# B&R Automation Studio project Ampel (part 2)

```cpp
	if (request.destination == 0)
		return false;
	else if (HFSM2_CHECKED(request.destination < STATE_COUNT)) {
Parent parent = stateParents[request.destination];

		if (HFSM2_CHECKED(parent)) {
			HFSM2_ASSERT(parent.forkId > 0);

compoRequested[parent.forkId - 1] = parent.prong;

for (parent = forkParent(parent.forkId);
parent;
parent = forkParent(parent.forkId))
			{
				HFSM2_ASSERT(parent.forkId > 0);
				compoRemains.set(parent.forkId - 1);

if (compoActive	  [parent.forkId - 1] != parent.prong)
compoRequested[parent.forkId - 1]  = parent.prong;
				else {
parent = forkParent(parent.forkId);
					break;
				}
			}

for (; parent; parent = forkParent(parent.forkId)) {
				HFSM2_ASSERT(parent.forkId > 0);
				compoRemains.set(parent.forkId - 1);
			}
		}
	}

	return true;
}

template <typename TG_, typename TSL_, typename TRL_, Long NCC_, typename TRO_ HFSM2_IF_SERIALIZATION(, Long NSB_) HFSM2_IF_PLANS(, Long NTC_), typename TTP_>
HFSM2_CONSTEXPR(14)
void
RegistryT<ArgsT<TG_, TSL_, TRL_, NCC_, 0, 0, TRO_ HFSM2_IF_SERIALIZATION(, NSB_) HFSM2_IF_PLANS(, NTC_), TTP_>>::requestScheduled(const StateID stateId) noexcept {
	if (HFSM2_CHECKED(stateId < STATE_COUNT)) {
const Parent parent = stateParents[stateId];

		HFSM2_ASSERT(parent.forkId > 0);
compoResumable[parent.forkId - 1] = parent.prong;
	}
}

template <typename TG_, typename TSL_, typename TRL_, Long NCC_, typename TRO_ HFSM2_IF_SERIALIZATION(, Long NSB_) HFSM2_IF_PLANS(, Long NTC_), typename TTP_>
HFSM2_CONSTEXPR(14)
void
RegistryT<ArgsT<TG_, TSL_, TRL_, NCC_, 0, 0, TRO_ HFSM2_IF_SERIALIZATION(, NSB_) HFSM2_IF_PLANS(, NTC_), TTP_>>::clearRequests() noexcept {
	compoRequested.clear();
	orthoRequested.clear();
	compoRemains  .clear();
}

template <typename TG_, typename TSL_, typename TRL_, Long NCC_, typename TRO_ HFSM2_IF_SERIALIZATION(, Long NSB_) HFSM2_IF_PLANS(, Long NTC_), typename TTP_>
HFSM2_CONSTEXPR(14)
void
RegistryT<ArgsT<TG_, TSL_, TRL_, NCC_, 0, 0, TRO_ HFSM2_IF_SERIALIZATION(, NSB_) HFSM2_IF_PLANS(, NTC_), TTP_>>::clear() noexcept {
	clearRequests();

	compoActive	  .clear();
	compoResumable.clear();
}

template <typename TG_, typename TSL_, typename TRL_, Long NCC_, typename TRO_ HFSM2_IF_SERIALIZATION(, Long NSB_) HFSM2_IF_PLANS(, Long NTC_), typename TTP_>
HFSM2_CONSTEXPR(11)
bool
RegistryT<ArgsT<TG_, TSL_, TRL_, NCC_, 0, 0, TRO_ HFSM2_IF_SERIALIZATION(, NSB_) HFSM2_IF_PLANS(, NTC_), TTP_>>::empty() const noexcept {
	return compoRequested.empty()
		&& orthoRequested.empty()
		&& compoRemains	 .empty()
		&& compoActive	 .empty()
		&& compoResumable.empty();
}

}
}

namespace hfsm2 {
	namespace detail {

		struct TaskStatus final {
		enum Result {
			NONE,
			SUCCESS,
			FAILURE
		};

		Result result = Result::NONE;
		bool outerTransition = false;

		HFSM2_CONSTEXPR(11)	TaskStatus(const Result result_ = Result::NONE,
		const bool outerTransition_ = false)	noexcept;

		HFSM2_CONSTEXPR(11)	explicit operator bool()				  const noexcept;

		HFSM2_CONSTEXPR(14)	void clear()									noexcept;
	};

	HFSM2_CONSTEXPR(14) TaskStatus  operator |  (TaskStatus& l, const TaskStatus r)	noexcept;
	HFSM2_CONSTEXPR(14) TaskStatus& operator |= (TaskStatus& l, const TaskStatus r)	noexcept;

#if HFSM2_PLANS_AVAILABLE()

	struct TaskLink final {
	Long prev		= INVALID_LONG;
	Long next		= INVALID_LONG;
};

struct Bounds final {
Long first		= INVALID_LONG;
Long last		= INVALID_LONG;
};

template <
	typename
  , typename
  , typename
  , Long
  , Long
  , Long
  , typename
  HFSM2_IF_SERIALIZATION(, Long)
, Long
  , typename
>
struct ArgsT;

template <typename>
struct PlanDataT;

template <
	typename TConfig
  , typename TStateList
  , typename TRegionList
  , Long NCompoCount
  , Long NOrthoCount
  , Long NOrthoUnits
  , typename TReactOrder
  HFSM2_IF_SERIALIZATION(, Long NSerialBits)
  , Long NTaskCapacity
  , typename TPayload
>
struct PlanDataT<
	ArgsT<
	TConfig
	, TStateList
	, TRegionList
	, NCompoCount
	, NOrthoCount
	, NOrthoUnits
	, TReactOrder
	HFSM2_IF_SERIALIZATION(, NSerialBits)
	, NTaskCapacity
	, TPayload
	>
	> final
	{
	using StateList			= TStateList;
	using RegionList		= TRegionList;
	using Payload			= TPayload;

	static constexpr Long STATE_COUNT	= StateList ::SIZE;
	static constexpr Long REGION_COUNT	= RegionList::SIZE;
	static constexpr Long TASK_CAPACITY	= NTaskCapacity;

	using Task				= TaskT		  <Payload>;
	using Tasks				= TaskListT   <Payload,  TASK_CAPACITY>;
	using TaskLinks			= StaticArrayT<TaskLink, TASK_CAPACITY>;
	using Payloads			= StaticArrayT<Payload,  TASK_CAPACITY>;

	using TasksBounds		= StaticArrayT<Bounds,	   REGION_COUNT>;
	using TasksBits			= BitArrayT   <				STATE_COUNT>;
	using RegionBits		= BitArrayT   <			   REGION_COUNT>;
	using RegionStatuses	= StaticArrayT<TaskStatus, REGION_COUNT>;

	Tasks tasks;
	TaskLinks taskLinks;
	Payloads taskPayloads;
	TasksBits payloadExists;

	TasksBounds taskBounds;
	TasksBits tasksSuccesses;
	TasksBits tasksFailures;
	RegionBits planExists;
	RegionStatuses headStatuses;
	RegionStatuses subStatuses;

	HFSM2_CONSTEXPR(14)	void clearTaskStatus  (const StateID stateId)		noexcept;
	HFSM2_CONSTEXPR(14)	void verifyEmptyStatus(const StateID stateId) const noexcept;

	HFSM2_CONSTEXPR(14)	void clearStatuses()								noexcept;
	HFSM2_CONSTEXPR(14)	void clear()										noexcept;

#if HFSM2_ASSERT_AVAILABLE()
	HFSM2_CONSTEXPR(14)	void verifyPlans()							  const noexcept;
	HFSM2_CONSTEXPR(14)	Long verifyPlan(const RegionID stateId)		  const noexcept;
#endif
};

template <
	typename TConfig
  , typename TStateList
  , typename TRegionList
  , Long NCompoCount
  , Long NOrthoCount
  , Long NOrthoUnits
  , typename TReactOrder
  HFSM2_IF_SERIALIZATION(, Long NSerialBits)
  , Long NTaskCapacity
>
struct PlanDataT<
		   ArgsT<
			   TConfig
			 , TStateList
			 , TRegionList
			 , NCompoCount
			 , NOrthoCount
			 , NOrthoUnits
			 , TReactOrder
			 HFSM2_IF_SERIALIZATION(, NSerialBits)
			 , NTaskCapacity
			 , void
		   >
	   > final
{
	using StateList			= TStateList;
using RegionList		= TRegionList;

static constexpr Long  STATE_COUNT	= StateList ::SIZE;
static constexpr Long REGION_COUNT	= RegionList::SIZE;
static constexpr Long TASK_CAPACITY	= NTaskCapacity;

	using Task				= TaskT		  <void>;
using Tasks				= TaskListT	  <void,	 TASK_CAPACITY>;
using TaskLinks			= StaticArrayT<TaskLink, TASK_CAPACITY>;

using TasksBounds		= StaticArrayT<Bounds,	   REGION_COUNT>;
using TasksBits			= BitArrayT	  <				STATE_COUNT>;
using RegionBits		= BitArrayT	  <			   REGION_COUNT>;
using RegionStatuses	= StaticArrayT<TaskStatus, REGION_COUNT>;

Tasks tasks;
TaskLinks taskLinks;

TasksBounds taskBounds;
TasksBits tasksSuccesses;
TasksBits tasksFailures;
RegionBits planExists;
RegionStatuses headStatuses;
RegionStatuses subStatuses;

	HFSM2_CONSTEXPR(14)	void clearTaskStatus  (const StateID stateId)		noexcept;
	HFSM2_CONSTEXPR(14)	void verifyEmptyStatus(const StateID stateId) const noexcept;

	HFSM2_CONSTEXPR(14)	void clearStatuses()								noexcept;
	HFSM2_CONSTEXPR(14)	void clear()										noexcept;

#if HFSM2_ASSERT_AVAILABLE()
	HFSM2_CONSTEXPR(14)	void verifyPlans()							  const noexcept;
	HFSM2_CONSTEXPR(14)	Long verifyPlan(const RegionID stateId)		  const noexcept;
#endif
};

template <
	typename TConfig
  , typename TStateList
  , typename TRegionList
  , Long NOrthoCount
  , Long NOrthoUnits
  , typename TReactOrder
  , Long NTaskCapacity
  , typename TPayload
>
struct PlanDataT<
	ArgsT<
	TConfig
	, TStateList
	, TRegionList
	, 0
	, NOrthoCount
	, NOrthoUnits
	, TReactOrder
	HFSM2_IF_SERIALIZATION(, 0)
	, NTaskCapacity
	, TPayload
	>
	> final
	{
HFSM2_CONSTEXPR(14)	void clearTaskStatus  (const StateID)				noexcept	{}
	HFSM2_CONSTEXPR(14)	void verifyEmptyStatus(const StateID)		  const noexcept	{}

	HFSM2_CONSTEXPR(14)	void clearStatuses()								noexcept	{}
	HFSM2_CONSTEXPR(14)	void clear()										noexcept	{}

#if HFSM2_ASSERT_AVAILABLE()
	HFSM2_CONSTEXPR(14)	void verifyPlans()							  const noexcept	{}
#endif
};

template <
	typename TConfig
  , typename TStateList
  , typename TRegionList
  , Long NOrthoCount
  , Long NOrthoUnits
  , typename TReactOrder
  , Long NTaskCapacity
>
struct PlanDataT<
		   ArgsT<
			   TConfig
			 , TStateList
			 , TRegionList
			 , 0
			 , NOrthoCount
			 , NOrthoUnits
			 , TReactOrder
			 HFSM2_IF_SERIALIZATION(, 0)
			 , NTaskCapacity
			 , void
		   >
	   > final
{
	HFSM2_CONSTEXPR(14)	void clearTaskStatus  (const StateID)				noexcept	{}
	HFSM2_CONSTEXPR(14)	void verifyEmptyStatus(const StateID)		  const noexcept	{}

	HFSM2_CONSTEXPR(14)	void clearStatuses()								noexcept	{}
	HFSM2_CONSTEXPR(14)	void clear()										noexcept	{}

#if HFSM2_ASSERT_AVAILABLE()
	HFSM2_CONSTEXPR(14)	void verifyPlans()							  const noexcept	{}
#endif
};

#endif

}
}

namespace hfsm2 {
	namespace detail {

		HFSM2_CONSTEXPR(11)
		TaskStatus::TaskStatus(const Result result_,
		const bool outerTransition_) noexcept
	: result{result_}
, outerTransition{outerTransition_}
{}

HFSM2_CONSTEXPR(11)
TaskStatus::operator bool() const noexcept	{
return result != Result::NONE || outerTransition;
}

HFSM2_CONSTEXPR(14)
void
TaskStatus::clear() noexcept {
result = Result::NONE;
outerTransition = false;
}

HFSM2_CONSTEXPR(14)
TaskStatus
	operator | (TaskStatus& lhs,
	const TaskStatus rhs) noexcept
{
	const TaskStatus::Result result = lhs.result > rhs.result ?
		lhs.result : rhs.result;

	return TaskStatus{result, lhs.outerTransition || rhs.outerTransition};
}

HFSM2_CONSTEXPR(14)
TaskStatus&
	operator |= (TaskStatus& lhs,
	const TaskStatus rhs) noexcept
{
	const TaskStatus::Result result = lhs.result > rhs.result ?
		lhs.result : rhs.result;

	lhs = TaskStatus{result, lhs.outerTransition || rhs.outerTransition};

	return lhs;
}

#if HFSM2_PLANS_AVAILABLE()

template <typename TG_, typename TSL_, typename TRL_, Long NCC_, Long NOC_, Long NOU_, typename TRO_ HFSM2_IF_SERIALIZATION(, Long NSB_), Long NTC_, typename TTP_>
HFSM2_CONSTEXPR(14)
void
	PlanDataT<ArgsT<TG_, TSL_, TRL_, NCC_, NOC_, NOU_, TRO_ HFSM2_IF_SERIALIZATION(, NSB_), NTC_, TTP_>>::clearTaskStatus(const StateID stateId) noexcept {
	if (stateId != INVALID_STATE_ID) {
		tasksSuccesses.clear(stateId);
		tasksFailures .clear(stateId);
	}
}

template <typename TG_, typename TSL_, typename TRL_, Long NCC_, Long NOC_, Long NOU_, typename TRO_ HFSM2_IF_SERIALIZATION(, Long NSB_), Long NTC_, typename TTP_>
HFSM2_CONSTEXPR(14)
void
	PlanDataT<ArgsT<TG_, TSL_, TRL_, NCC_, NOC_, NOU_, TRO_ HFSM2_IF_SERIALIZATION(, NSB_), NTC_, TTP_>>::verifyEmptyStatus(const StateID HFSM2_IF_ASSERT(stateId)) const noexcept {
#if HFSM2_ASSERT_AVAILABLE()

	if (stateId != INVALID_STATE_ID) {
		HFSM2_ASSERT(!tasksSuccesses.get(stateId));
		HFSM2_ASSERT(!tasksFailures .get(stateId));
	}

#endif
}

template <typename TG_, typename TSL_, typename TRL_, Long NCC_, Long NOC_, Long NOU_, typename TRO_ HFSM2_IF_SERIALIZATION(, Long NSB_), Long NTC_, typename TTP_>
HFSM2_CONSTEXPR(14)
void
	PlanDataT<ArgsT<TG_, TSL_, TRL_, NCC_, NOC_, NOU_, TRO_ HFSM2_IF_SERIALIZATION(, NSB_), NTC_, TTP_>>::clearStatuses() noexcept {
	tasksSuccesses.clear();
	tasksFailures .clear();

	headStatuses.clear();
	 subStatuses.clear();
}

template <typename TG_, typename TSL_, typename TRL_, Long NCC_, Long NOC_, Long NOU_, typename TRO_ HFSM2_IF_SERIALIZATION(, Long NSB_), Long NTC_, typename TTP_>
HFSM2_CONSTEXPR(14)
void
	PlanDataT<ArgsT<TG_, TSL_, TRL_, NCC_, NOC_, NOU_, TRO_ HFSM2_IF_SERIALIZATION(, NSB_), NTC_, TTP_>>::clear() noexcept {
	tasks		 .clear();
	taskLinks	 .clear();
	taskPayloads .clear();
	payloadExists.clear();

	taskBounds	 .clear();
	planExists	 .clear();

	clearStatuses();
}

#if HFSM2_ASSERT_AVAILABLE()

template <typename TG_, typename TSL_, typename TRL_, Long NCC_, Long NOC_, Long NOU_, typename TRO_ HFSM2_IF_SERIALIZATION(, Long NSB_), Long NTC_, typename TTP_>
HFSM2_CONSTEXPR(14)
void
	PlanDataT<ArgsT<TG_, TSL_, TRL_, NCC_, NOC_, NOU_, TRO_ HFSM2_IF_SERIALIZATION(, NSB_), NTC_, TTP_>>::verifyPlans() const noexcept {
Long planCount = 0;

for (RegionID regionId = 0; regionId < REGION_COUNT; ++regionId)
		planCount += verifyPlan(regionId);

	HFSM2_ASSERT(tasks.count() == planCount);
}

template <typename TG_, typename TSL_, typename TRL_, Long NCC_, Long NOC_, Long NOU_, typename TRO_ HFSM2_IF_SERIALIZATION(, Long NSB_), Long NTC_, typename TTP_>
HFSM2_CONSTEXPR(14)
Long
	PlanDataT<ArgsT<TG_, TSL_, TRL_, NCC_, NOC_, NOU_, TRO_ HFSM2_IF_SERIALIZATION(, NSB_), NTC_, TTP_>>::verifyPlan(const RegionID regionId) const noexcept {
Long length = 0;
const Bounds& bounds = taskBounds[regionId];

	if (bounds.first != INVALID_LONG) {
		HFSM2_ASSERT(bounds.last != INVALID_LONG);

for (Long slow = bounds.first, fast = slow; ; ) {
++length;
const TaskLink& task = taskLinks[slow];

			if (slow != bounds.last) {
				HFSM2_ASSERT(task.next != INVALID_LONG);
slow = task.next;

				// loop check
				if (fast != INVALID_LONG) {
fast = taskLinks[fast].next;

					if (fast != INVALID_LONG)
fast = taskLinks[fast].next;

					HFSM2_ASSERT(fast == INVALID_LONG || slow != fast);
				}
			} else {
				HFSM2_ASSERT(task.next == INVALID_LONG);

				break;
			}
		};
	} else
		HFSM2_ASSERT(bounds.last == INVALID_LONG);

return length;
}

#endif

template <typename TG_, typename TSL_, typename TRL_, Long NCC_, Long NOC_, Long NOU_, typename TRO_ HFSM2_IF_SERIALIZATION(, Long NSB_), Long NTC_>
HFSM2_CONSTEXPR(14)
void
PlanDataT<ArgsT<TG_, TSL_, TRL_, NCC_, NOC_, NOU_, TRO_ HFSM2_IF_SERIALIZATION(, NSB_), NTC_, void>>::clearTaskStatus(const StateID stateId) noexcept {
	if (stateId != INVALID_STATE_ID) {
		tasksSuccesses.clear(stateId);
		tasksFailures .clear(stateId);
	}
}

template <typename TG_, typename TSL_, typename TRL_, Long NCC_, Long NOC_, Long NOU_, typename TRO_ HFSM2_IF_SERIALIZATION(, Long NSB_), Long NTC_>
HFSM2_CONSTEXPR(14)
void
PlanDataT<ArgsT<TG_, TSL_, TRL_, NCC_, NOC_, NOU_, TRO_ HFSM2_IF_SERIALIZATION(, NSB_), NTC_, void>>::verifyEmptyStatus(const StateID HFSM2_IF_ASSERT(stateId)) const noexcept {
#if HFSM2_ASSERT_AVAILABLE()

	if (stateId != INVALID_STATE_ID) {
		HFSM2_ASSERT(!tasksSuccesses.get(stateId));
		HFSM2_ASSERT(!tasksFailures .get(stateId));
	}

#endif
}

template <typename TG_, typename TSL_, typename TRL_, Long NCC_, Long NOC_, Long NOU_, typename TRO_ HFSM2_IF_SERIALIZATION(, Long NSB_), Long NTC_>
HFSM2_CONSTEXPR(14)
void
PlanDataT<ArgsT<TG_, TSL_, TRL_, NCC_, NOC_, NOU_, TRO_ HFSM2_IF_SERIALIZATION(, NSB_), NTC_, void>>::clearStatuses() noexcept {
	tasksSuccesses.clear();
	tasksFailures .clear();

	headStatuses.clear();
	 subStatuses.clear();
}

template <typename TG_, typename TSL_, typename TRL_, Long NCC_, Long NOC_, Long NOU_, typename TRO_ HFSM2_IF_SERIALIZATION(, Long NSB_), Long NTC_>
HFSM2_CONSTEXPR(14)
void
PlanDataT<ArgsT<TG_, TSL_, TRL_, NCC_, NOC_, NOU_, TRO_ HFSM2_IF_SERIALIZATION(, NSB_), NTC_, void>>::clear() noexcept {
	tasks	  .clear();
	taskLinks .clear();

	taskBounds.clear();
	planExists.clear();

	clearStatuses();
}

#if HFSM2_ASSERT_AVAILABLE()

template <typename TG_, typename TSL_, typename TRL_, Long NCC_, Long NOC_, Long NOU_, typename TRO_ HFSM2_IF_SERIALIZATION(, Long NSB_), Long NTC_>
HFSM2_CONSTEXPR(14)
void
PlanDataT<ArgsT<TG_, TSL_, TRL_, NCC_, NOC_, NOU_, TRO_ HFSM2_IF_SERIALIZATION(, NSB_), NTC_, void>>::verifyPlans() const noexcept {
Long planCount = 0;

for (RegionID regionId = 0; regionId < REGION_COUNT; ++regionId)
		planCount += verifyPlan(regionId);

	HFSM2_ASSERT(tasks.count() == planCount);
}

template <typename TG_, typename TSL_, typename TRL_, Long NCC_, Long NOC_, Long NOU_, typename TRO_ HFSM2_IF_SERIALIZATION(, Long NSB_), Long NTC_>
HFSM2_CONSTEXPR(14)
Long
PlanDataT<ArgsT<TG_, TSL_, TRL_, NCC_, NOC_, NOU_, TRO_ HFSM2_IF_SERIALIZATION(, NSB_), NTC_, void>>::verifyPlan(const RegionID regionId) const noexcept {
Long length = 0;
const Bounds& bounds = taskBounds[regionId];

	if (bounds.first != INVALID_LONG) {
		HFSM2_ASSERT(bounds.last != INVALID_LONG);

for (auto slow = bounds.first, fast = slow; ; ) {
++length;
const TaskLink& task = taskLinks[slow];

			if (slow != bounds.last) {
				HFSM2_ASSERT(task.next != INVALID_LONG);
slow = task.next;

				// loop check
				if (fast != INVALID_LONG) {
fast = taskLinks[fast].next;

					if (fast != INVALID_LONG)
fast = taskLinks[fast].next;

					HFSM2_ASSERT(fast == INVALID_LONG || slow != fast);
				}
			} else {
				HFSM2_ASSERT(task.next == INVALID_LONG);

				break;
			}
		};
	} else
		HFSM2_ASSERT(bounds.last == INVALID_LONG);

return length;
}

#endif
#endif

}
}

#if HFSM2_PLANS_AVAILABLE()

namespace hfsm2 {
	namespace detail {

		template <typename TArgs>
		class CPlanT {
			template <typename>
			friend class ControlT;

			template <typename>
			friend class PlanControlT;

			template <typename>
			friend class FullControlT;

			template <typename>
			friend class GuardControlT;

			template <typename, typename>
			friend class R_;

			using Args			= TArgs;
			using Context		= typename Args::Context;
			using StateList		= typename Args::StateList;
			using RegionList	= typename Args::RegionList;

			static constexpr Long TASK_CAPACITY = Args::TASK_CAPACITY;

			public:
			using PlanData		= PlanDataT<Args>;
			using Task			= typename PlanData::Task;
			using TaskLinks		= typename PlanData::TaskLinks;

			struct Iterator final {
			HFSM2_CONSTEXPR(14)	Iterator(const CPlanT& plan)				noexcept;

			HFSM2_CONSTEXPR(14)	explicit operator bool()			  const noexcept;

			HFSM2_CONSTEXPR(14)	void operator ++()							noexcept;

			HFSM2_CONSTEXPR(11)	bool operator != (const Iterator)	  const noexcept	{ return operator bool();					}

			HFSM2_CONSTEXPR(11)	const Task& operator  *()			  const noexcept	{ return  _plan._planData.tasks[_curr];		}
			HFSM2_CONSTEXPR(11)	const Task* operator ->()			  const noexcept	{ return &_plan._planData.tasks[_curr];		}

			HFSM2_CONSTEXPR(14)	Long next()							  const noexcept;

			const CPlanT& _plan;
			Long _curr;
			Long _next;
		};

		private:
		HFSM2_CONSTEXPR(11)	CPlanT(const PlanData& planData,
		const RegionID regionId_)				noexcept
	: _planData{planData}
, _bounds{planData.taskBounds[regionId_]}
	{}

	template <typename TState>
	static
	HFSM2_CONSTEXPR(11)  StateID  stateId()								noexcept	{ return					   index<StateList , TState>();		}

	template <typename TState>
	static
	HFSM2_CONSTEXPR(11)	RegionID regionId()								noexcept	{ return static_cast<RegionID>(index<RegionList, TState>());	}

public:
	HFSM2_CONSTEXPR(14)	explicit operator bool()				  const noexcept;

	/// @brief Begin iteration over plan tasks
	/// @return CIterator to the first task
	HFSM2_CONSTEXPR(14)	Iterator begin()								noexcept	{ return Iterator{*this};					}

	/// @brief Iteration terminator
	/// @return Dummy Iterator
	HFSM2_CONSTEXPR(14)	Iterator end  ()								noexcept	{ return Iterator{*this};					}

	/// @brief First task
	/// @return First task
	HFSM2_CONSTEXPR(14) const Task& first()						  const noexcept;

	/// @brief Last task
	/// @return Last task
	HFSM2_CONSTEXPR(14) const Task&  last()						  const noexcept;

private:
const PlanData& _planData;
const Bounds& _bounds;
};

}
}

#endif

#if HFSM2_PLANS_AVAILABLE()

namespace hfsm2 {
	namespace detail {

		template <typename TArgs>
		HFSM2_CONSTEXPR(14)
		CPlanT<TArgs>::Iterator::Iterator(const CPlanT& plan) noexcept
	: _plan{plan}
, _curr{plan._bounds.first}
{
	_next = next();
}

template <typename TArgs>
HFSM2_CONSTEXPR(14)
CPlanT<TArgs>::Iterator::operator bool() const noexcept {
	HFSM2_ASSERT(_curr < CPlanT::TASK_CAPACITY ||
				 _curr == INVALID_LONG);

return _curr < CPlanT::TASK_CAPACITY;
}

template <typename TArgs>
HFSM2_CONSTEXPR(14)
void
CPlanT<TArgs>::Iterator::operator ++() noexcept {
	_curr = _next;
	_next = next();
}

template <typename TArgs>
HFSM2_CONSTEXPR(14)
Long
CPlanT<TArgs>::Iterator::next() const noexcept {
	if (_curr < CPlanT::TASK_CAPACITY) {
		const TaskLink& link = _plan._planData.taskLinks[_curr];

		return link.next;
	} else {
		HFSM2_ASSERT(_curr == INVALID_LONG);

		return INVALID_LONG;
	}
}

template <typename TArgs>
HFSM2_CONSTEXPR(14)
CPlanT<TArgs>::operator bool() const noexcept {
	HFSM2_ASSERT(_bounds.first < TASK_CAPACITY &&
				 _bounds.last  < TASK_CAPACITY ||
				 _bounds.last == INVALID_LONG);

return _bounds.first < TASK_CAPACITY;
}

template <typename TArgs>
HFSM2_CONSTEXPR(14)
const typename CPlanT<TArgs>::Task&
CPlanT<TArgs>::first() const noexcept {
	HFSM2_ASSERT(_bounds.first < TASK_CAPACITY);

	return _planData.tasks[_bounds.first];
}

template <typename TArgs>
HFSM2_CONSTEXPR(14)
const typename CPlanT<TArgs>::Task&
CPlanT<TArgs>::last() const noexcept {
	HFSM2_ASSERT(_bounds.last < TASK_CAPACITY);

	return _planData.tasks[_bounds.last];
}

}
}

#endif

#if HFSM2_PLANS_AVAILABLE()

namespace hfsm2 {
	namespace detail {

		template <typename TArgs>
		class PlanT {
			template <typename, typename, Strategy, typename, typename...>
			friend struct C_;

			template <typename, typename, typename, typename...>
			friend struct O_;

			using Args			= TArgs;
			using Context		= typename Args::Context;
			using StateList		= typename Args::StateList;
			using RegionList	= typename Args::RegionList;

			using Registry		= RegistryT<Args>;

			static constexpr Long  TASK_CAPACITY	= Args::TASK_CAPACITY;

			public:
			using PlanData		= PlanDataT<Args>;
			using Task			= typename PlanData::Task;
			using Tasks			= typename PlanData::Tasks;
			using TaskLinks		= typename PlanData::TaskLinks;
			using TaskIndex		= typename TaskLinks::Index;
			using TasksBits		= typename PlanData::TasksBits;

			struct CIterator final {
			HFSM2_CONSTEXPR(14)	CIterator(const PlanT& plan)				noexcept;

			HFSM2_CONSTEXPR(14)	explicit operator bool()			  const noexcept;

			HFSM2_CONSTEXPR(14)	void operator ++()							noexcept;

			HFSM2_CONSTEXPR(14)	bool operator != (const CIterator)	  const noexcept	{ return operator bool();					}

			HFSM2_CONSTEXPR(14)	const Task& operator  *()			  const noexcept	{ return  _plan._planData.tasks[_curr];		}
			HFSM2_CONSTEXPR(11)	const Task* operator ->()			  const noexcept	{ return &_plan._planData.tasks[_curr];		}

			HFSM2_CONSTEXPR(14)	Long next()							  const noexcept;

			const PlanT& _plan;
			Long _curr;
			Long _next;
		};

		struct Iterator final {
		HFSM2_CONSTEXPR(14)	Iterator(PlanT& plan)						noexcept;

		HFSM2_CONSTEXPR(14)	explicit operator bool()			  const noexcept;

		HFSM2_CONSTEXPR(14)	void operator ++()							noexcept;

		HFSM2_CONSTEXPR(14)	bool operator != (const Iterator)	  const noexcept	{ return operator bool();					}

		HFSM2_CONSTEXPR(14)	Task& operator  *()							noexcept	{ return  _plan._planData.tasks[_curr];		}
		HFSM2_CONSTEXPR(14)	Task* operator ->()							noexcept	{ return &_plan._planData.tasks[_curr];		}

	HFSM2_CONSTEXPR(14)	void remove()								noexcept	{ _plan.remove(_curr);						}

	HFSM2_CONSTEXPR(14)	Long next()							  const noexcept;

	PlanT& _plan;
	Long _curr;
	Long _next;
};

protected:
	HFSM2_CONSTEXPR(11)	PlanT(Registry& registry,
							  PlanData& planData,
							  const RegionID regionId_)					noexcept;

	template <typename TState>
	static
	HFSM2_CONSTEXPR(11)  StateID  stateId()								noexcept	{ return					   index<StateList , TState>();		}

	template <typename TState>
	static
	HFSM2_CONSTEXPR(11) RegionID regionId()								noexcept	{ return static_cast<RegionID>(index<RegionList, TState>());	}

	HFSM2_CONSTEXPR(14)	bool  append(const StateID origin,
									 const StateID destination,
									 const TransitionType type)			noexcept;

	HFSM2_CONSTEXPR(14)	bool linkTask(const Long index)					noexcept;

	HFSM2_CONSTEXPR(14)	void clearTasks()								noexcept;
	HFSM2_CONSTEXPR(14)	void clearStatuses()							noexcept;

public:
	HFSM2_CONSTEXPR(14)	explicit operator bool()				  const noexcept;

	/// @brief Clear all tasks from the plan
	HFSM2_CONSTEXPR(14)	void clear()									noexcept;

	/// @brief Append a task to transition from `origin` to `destination` if `origin` completes with `success()`
	///   (if transitioning into a region, acts depending on the region type)
	/// @param `origin` Origin state identifier
	/// @param `destination` Destination state identifier
	/// @return Seccess if FSM total number of tasks is below task capacity
	/// @note use `Config::TaskCapacityN<>` to increase task capacity if necessary
	HFSM2_CONSTEXPR(14)	bool change   (const StateID origin,
									   const StateID destination)		noexcept	{ return append	  (origin, destination, TransitionType::CHANGE	 );	}

	/// @brief Append a task to transition from `origin` to `destination` if `origin` completes with `success()`
	///   (if transitioning into a region, acts depending on the region type)
	/// @tparam `TOrigin` Origin state type
	/// @param `destination` Destination state identifier
	/// @return Seccess if FSM total number of tasks is below task capacity
	/// @note use `Config::TaskCapacityN<>` to increase task capacity if necessary
	template <typename TOrigin>
	HFSM2_CONSTEXPR(14)	bool change   (const StateID destination)		noexcept	{ return change	  (stateId<TOrigin>() , destination				 );	}

	/// @brief Append a task to transition from `origin` to `destination` if `origin` completes with `success()`
	///   (if transitioning into a region, acts depending on the region type)
	/// @tparam `TOrigin` Origin state type
	/// @tparam `TDestination` Destination state type
	/// @return Seccess if FSM total number of tasks is below task capacity
	/// @note use `Config::TaskCapacityN<>` to increase task capacity if necessary
	template <typename TOrigin, typename TDestination>
	HFSM2_CONSTEXPR(14)	bool change   ()								noexcept	{ return change	  (stateId<TOrigin>() , stateId<TDestination>()	 );	}

	/// @brief Append a task to transition from `origin` to `destination` if `origin` completes with `success()`
	///   (if transitioning into a region, activates the initial state)
	/// @tparam `TOrigin` Origin state type
	/// @param `destination` Destination state identifier
	/// @return Seccess if FSM total number of tasks is below task capacity
	/// @note use `Config::TaskCapacityN<>` to increase task capacity if necessary
	HFSM2_CONSTEXPR(14)	bool restart  (const StateID origin,
									   const StateID destination)		noexcept	{ return append	  (origin, destination, TransitionType::RESTART	 );	}

	/// @brief Append a task to transition from `origin` to `destination` if `origin` completes with `success()`
	///   (if transitioning into a region, activates the initial state)
	/// @tparam `TOrigin` Origin state type
	/// @param `destination` Destination state identifier
	/// @return Seccess if FSM total number of tasks is below task capacity
	/// @note use `Config::TaskCapacityN<>` to increase task capacity if necessary
	template <typename TOrigin>
	HFSM2_CONSTEXPR(14)	bool restart  (const StateID destination)		noexcept	{ return restart  (stateId<TOrigin>() , destination				 );	}

	/// @brief Append a task to transition from `origin` to `destination` if `origin` completes with `success()`
	///   (if transitioning into a region, activates the initial state)
	/// @tparam `TOrigin` Origin state type
	/// @tparam `TDestination` Destination state type
	/// @return Seccess if FSM total number of tasks is below task capacity
	/// @note use `Config::TaskCapacityN<>` to increase task capacity if necessary
	template <typename TOrigin, typename TDestination>
	HFSM2_CONSTEXPR(14)	bool restart  ()								noexcept	{ return restart  (stateId<TOrigin>() , stateId<TDestination>()	 );	}

	/// @brief Append a task to transition from `origin` to `destination` if `origin` completes with `success()`
	///   (if transitioning into a region, activates the state that was active previously)
	/// @tparam `TOrigin` Origin state type
	/// @param `destination` Destination state identifier
	/// @return Seccess if FSM total number of tasks is below task capacity
	/// @note use `Config::TaskCapacityN<>` to increase task capacity if necessary
	HFSM2_CONSTEXPR(14)	bool resume   (const StateID origin,
									   const StateID destination)		noexcept	{ return append	  (origin, destination, TransitionType::RESUME	 );	}

	/// @brief Append a task to transition from `origin` to `destination` if `origin` completes with `success()`
	///   (if transitioning into a region, activates the state that was active previously)
	/// @tparam `TOrigin` Origin state type
	/// @param `destination` Destination state identifier
	/// @return Seccess if FSM total number of tasks is below task capacity
	/// @note use `Config::TaskCapacityN<>` to increase task capacity if necessary
	template <typename TOrigin>
	HFSM2_CONSTEXPR(14)	bool resume   (const StateID destination)		noexcept	{ return resume	  (stateId<TOrigin>() , destination				 );	}

	/// @brief Append a task to transition from `origin` to `destination` if `origin` completes with `success()`
	///   (if transitioning into a region, activates the state that was active previously)
	/// @tparam `TOrigin` Origin state type
	/// @tparam `TDestination` Destination state type
	/// @return Seccess if FSM total number of tasks is below task capacity
	/// @note use `Config::TaskCapacityN<>` to increase task capacity if necessary
	template <typename TOrigin, typename TDestination>
	HFSM2_CONSTEXPR(14)	bool resume   ()								noexcept	{ return resume	  (stateId<TOrigin>() , stateId<TDestination>()	 );	}

	/// @brief Append a task to transition from `origin` to `destination` if `origin` completes with `success()`
	///   (if transitioning into a region, activates the sub-state by index returned by the region's `select()` method)
	/// @tparam `TOrigin` Origin state type
	/// @param `destination` Destination state identifier
	/// @return Seccess if FSM total number of tasks is below task capacity
	/// @note use `Config::TaskCapacityN<>` to increase task capacity if necessary
	HFSM2_CONSTEXPR(14)	bool select   (const StateID origin,
									   const StateID destination)		noexcept	{ return append	  (origin, destination, TransitionType::SELECT	 );	}

	/// @brief Append a task to transition from `origin` to `destination` if `origin` completes with `success()`
	///   (if transitioning into a region, activates the sub-state by index returned by the region's `select()` method)
	/// @tparam `TOrigin` Origin state type
	/// @param `destination` Destination state identifier
	/// @return Seccess if FSM total number of tasks is below task capacity
	/// @note use `Config::TaskCapacityN<>` to increase task capacity if necessary
	template <typename TOrigin>
	HFSM2_CONSTEXPR(14)	bool select   (const StateID destination)		noexcept	{ return select	  (stateId<TOrigin>() , destination				 );	}

	/// @brief Append a task to transition from `origin` to `destination` if `origin` completes with `success()`
	///   (if transitioning into a region, activates the sub-state by index returned by the region's `select()` method)
	/// @tparam `TOrigin` Origin state type
	/// @tparam `TDestination` Destination state type
	/// @return Seccess if FSM total number of tasks is below task capacity
	/// @note use `Config::TaskCapacityN<>` to increase task capacity if necessary
	template <typename TOrigin, typename TDestination>
	HFSM2_CONSTEXPR(14)	bool select   ()								noexcept	{ return select	  (stateId<TOrigin>() , stateId<TDestination>()	 );	}

#if HFSM2_UTILITY_THEORY_AVAILABLE()

	/// @brief Append a task to transition from `origin` to `destination` if `origin` completes with `success()`
	///   (if transitioning into a region, activates the state with the highest `utility()`
	///   among those with the highest `rank()`)
	/// @tparam `TOrigin` Origin state type
	/// @param `destination` Destination state identifier
	/// @return Seccess if FSM total number of tasks is below task capacity
	/// @note use `Config::TaskCapacityN<>` to increase task capacity if necessary
	/// @see `HFSM2_ENABLE_UTILITY_THEORY`
	HFSM2_CONSTEXPR(14)	bool utilize  (const StateID origin,
									   const StateID destination)		noexcept	{ return append	  (origin, destination, TransitionType::UTILIZE	 );	}

	/// @brief Append a task to transition from `origin` to `destination` if `origin` completes with `success()`
	///   (if transitioning into a region, activates the state with the highest `utility()`
	///   among those with the highest `rank()`)
	/// @tparam `TOrigin` Origin state type
	/// @param `destination` Destination state identifier
	/// @return Seccess if FSM total number of tasks is below task capacity
	/// @note use `Config::TaskCapacityN<>` to increase task capacity if necessary
	/// @see `HFSM2_ENABLE_UTILITY_THEORY`
	template <typename TOrigin>
	HFSM2_CONSTEXPR(14)	bool utilize  (const StateID destination)		noexcept	{ return utilize  (stateId<TOrigin>() , destination				 );	}

	/// @brief Append a task to transition from `origin` to `destination` if `origin` completes with `success()`
	///   (if transitioning into a region, activates the state with the highest `utility()`
	///   among those with the highest `rank()`)
	/// @tparam `TOrigin` Origin state type
	/// @tparam `TDestination` Destination state type
	/// @return Seccess if FSM total number of tasks is below task capacity
	/// @note use `Config::TaskCapacityN<>` to increase task capacity if necessary
	/// @see `HFSM2_ENABLE_UTILITY_THEORY`
	template <typename TOrigin, typename TDestination>
	HFSM2_CONSTEXPR(14)	bool utilize  ()								noexcept	{ return utilize  (stateId<TOrigin>() , stateId<TDestination>()	 );	}

	/// @brief Append a task to transition from `origin` to `destination` if `origin` completes with `success()`
	///   (if transitioning into a region, uses weighted random to activate the state proportional to `utility()`
	///   among those with the highest `rank()`)
	/// @tparam `TOrigin` Origin state type
	/// @param `destination` Destination state identifier
	/// @return Seccess if FSM total number of tasks is below task capacity
	/// @note use `Config::TaskCapacityN<>` to increase task capacity if necessary
	/// @see `HFSM2_ENABLE_UTILITY_THEORY`
	HFSM2_CONSTEXPR(14)	bool randomize(const StateID origin,
									   const StateID destination)		noexcept	{ return append	  (origin, destination, TransitionType::RANDOMIZE);	}

	/// @brief Append a task to transition from `origin` to `destination` if `origin` completes with `success()`
	///   (if transitioning into a region, uses weighted random to activate the state proportional to `utility()`
	///   among those with the highest `rank()`)
	/// @tparam `TOrigin` Origin state type
	/// @param `destination` Destination state identifier
	/// @return Seccess if FSM total number of tasks is below task capacity
	/// @note use `Config::TaskCapacityN<>` to increase task capacity if necessary
	/// @see `HFSM2_ENABLE_UTILITY_THEORY`
	template <typename TOrigin>
	HFSM2_CONSTEXPR(14)	bool randomize(const StateID destination)		noexcept	{ return randomize(stateId<TOrigin>() , destination				 );	}

	/// @brief Append a task to transition from `origin` to `destination` if `origin` completes with `success()`
	///   (if transitioning into a region, uses weighted random to activate the state proportional to `utility()`
	///   among those with the highest `rank()`)
	/// @tparam `TOrigin` Origin state type
	/// @tparam `TDestination` Destination state type
	/// @return Seccess if FSM total number of tasks is below task capacity
	/// @note use `Config::TaskCapacityN<>` to increase task capacity if necessary
	/// @see `HFSM2_ENABLE_UTILITY_THEORY`
	template <typename TOrigin, typename TDestination>
	HFSM2_CONSTEXPR(14)	bool randomize()								noexcept	{ return randomize(stateId<TOrigin>() , stateId<TDestination>()	 );	}

#endif

	/// @brief Append a task to schedule a transition to `destination` if `origin` completes with `success()`
	/// @tparam `TOrigin` Origin state type
	/// @param `destination` Destination state identifier
	/// @return Seccess if FSM total number of tasks is below task capacity
	/// @note use `Config::TaskCapacityN<>` to increase task capacity if necessary
	HFSM2_CONSTEXPR(14)	bool schedule (const StateID origin,
									   const StateID destination)		noexcept	{ return append	  (origin, destination, TransitionType::SCHEDULE );	}

	/// @brief Append a task to schedule a transition to `destination` if `origin` completes with `success()`
	/// @tparam `TOrigin` Origin state type
	/// @param `destination` Destination state identifier
	/// @return Seccess if FSM total number of tasks is below task capacity
	/// @note use `Config::TaskCapacityN<>` to increase task capacity if necessary
	template <typename TOrigin>
	HFSM2_CONSTEXPR(14)	bool schedule (const StateID destination)		noexcept	{ return schedule (stateId<TOrigin>() , destination				 );	}

	/// @brief Append a task to schedule a transition to `destination` if `origin` completes with `success()`
	/// @tparam `TOrigin` Origin state type
	/// @tparam `TDestination` Destination state type
	/// @return Seccess if FSM total number of tasks is below task capacity
	/// @note use `Config::TaskCapacityN<>` to increase task capacity if necessary
	template <typename TOrigin, typename TDestination>
	HFSM2_CONSTEXPR(14)	bool schedule ()								noexcept	{ return schedule (stateId<TOrigin>() , stateId<TDestination>()	 );	}

	/// @brief Begin iteration over plan tasks
	/// @return Iterator to the first task
	HFSM2_CONSTEXPR(14)	 Iterator begin()								noexcept	{ return  Iterator{*this};	}

	/// @brief Begin iteration over plan tasks
	/// @return CIterator to the first task
	HFSM2_CONSTEXPR(11)	CIterator begin()						  const noexcept	{ return CIterator{*this};	}

private:
	HFSM2_CONSTEXPR(14)	void remove(const Long task)					noexcept;

protected:
Registry& _registry;
PlanData& _planData;
const RegionID _regionId;
Bounds& _bounds;
};

}
}

#endif

#if HFSM2_PLANS_AVAILABLE()

namespace hfsm2 {
	namespace detail {

		template <typename TArgs>
		HFSM2_CONSTEXPR(14)
		PlanT<TArgs>::CIterator::CIterator(const PlanT& plan) noexcept
	: _plan{plan}
, _curr{plan._bounds.first}
	, _next{next()}
{}

template <typename TArgs>
HFSM2_CONSTEXPR(14)
PlanT<TArgs>::CIterator::operator bool() const noexcept {
	HFSM2_ASSERT(_curr  < PlanT::TASK_CAPACITY ||
				 _curr == INVALID_LONG);

return _curr < PlanT::TASK_CAPACITY;
}

template <typename TArgs>
HFSM2_CONSTEXPR(14)
void
PlanT<TArgs>::CIterator::operator ++() noexcept {
	_curr = _next;
	_next = next();
}

template <typename TArgs>
HFSM2_CONSTEXPR(14)
Long
PlanT<TArgs>::CIterator::next() const noexcept {
	if (_curr < PlanT::TASK_CAPACITY) {
		const TaskLink& link = _plan._planData.taskLinks[_curr];

		return link.next;
	} else {
		HFSM2_ASSERT(_curr == INVALID_LONG);

		return INVALID_LONG;
	}
}

template <typename TArgs>
HFSM2_CONSTEXPR(14)
PlanT<TArgs>::Iterator::Iterator(PlanT& plan) noexcept
	: _plan{plan}
	, _curr{plan._bounds.first}
	, _next{next()}
{}

template <typename TArgs>
HFSM2_CONSTEXPR(14)
PlanT<TArgs>::Iterator::operator bool() const noexcept {
	HFSM2_ASSERT(_curr < PlanT::TASK_CAPACITY ||
				 _curr == INVALID_LONG);

return _curr < PlanT::TASK_CAPACITY;
}

template <typename TArgs>
HFSM2_CONSTEXPR(14)
void
PlanT<TArgs>::Iterator::operator ++() noexcept {
	_curr = _next;
	_next = next();
}

template <typename TArgs>
HFSM2_CONSTEXPR(14)
Long
PlanT<TArgs>::Iterator::next() const noexcept {
	if (_curr < PlanT::TASK_CAPACITY) {
		const TaskLink& link = _plan._planData.taskLinks[_curr];

		return link.next;
	} else {
		HFSM2_ASSERT(_curr == INVALID_LONG);

		return INVALID_LONG;
	}
}

template <typename TArgs>
HFSM2_CONSTEXPR(11)
PlanT<TArgs>::PlanT(Registry& registry,
					PlanData& planData,
					const RegionID regionId_) noexcept
	: _registry{registry}
	, _planData{planData}
	, _regionId{regionId_}
, _bounds{planData.taskBounds[regionId_]}
{}

template <typename TArgs>
HFSM2_CONSTEXPR(14)
bool
PlanT<TArgs>:: append(const StateID origin,
					  const StateID destination,
					  const TransitionType type) noexcept
{
	if (_planData.tasks.count() < TASK_CAPACITY) {
		_planData.planExists.set(_regionId);

		return linkTask(_planData.tasks.emplace(origin, destination, type));
	} else
		return false;
}

template <typename TArgs>
HFSM2_CONSTEXPR(14)
bool
PlanT<TArgs>::linkTask(const Long index) noexcept {
	if (index != Tasks::INVALID) {
		if (_bounds.first == INVALID_LONG) {
			HFSM2_ASSERT(_bounds.last == INVALID_LONG);
			HFSM2_ASSERT(_planData.taskLinks[index].prev == INVALID_LONG);
			HFSM2_ASSERT(_planData.taskLinks[index].next == INVALID_LONG);

_bounds.first = index;
_bounds.last  = index;
		} else {
			HFSM2_ASSERT(_bounds.first < TaskLinks::CAPACITY);
			HFSM2_ASSERT(_bounds.last  < TaskLinks::CAPACITY);

TaskLink& lastLink = _planData.taskLinks[_bounds.last];
			HFSM2_ASSERT(lastLink.next == INVALID_LONG);

lastLink.next  = index;

TaskLink& currLink = _planData.taskLinks[index];
			HFSM2_ASSERT(currLink.prev == INVALID_LONG);

currLink.prev  = _bounds.last;

_bounds.last   = index;
		}

		return true;
	} else
		return false;
}

template <typename TArgs>
HFSM2_CONSTEXPR(14)
void
PlanT<TArgs>::clearTasks() noexcept {
	if (_bounds.first < TaskLinks::CAPACITY) {
		HFSM2_ASSERT(_bounds.last < TaskLinks::CAPACITY);

for (Long index = _bounds.first;
index != INVALID_LONG;
			 )
		{
			HFSM2_ASSERT(index < TaskLinks::CAPACITY);

const TaskLink& link = _planData.taskLinks[index];
			HFSM2_ASSERT(index == _bounds.first ?
							 link.prev == INVALID_LONG :
							 link.prev <  TaskLinks::CAPACITY);

const Long next = link.next;

			remove(index);

index = next;
		}

_bounds.first = INVALID_LONG;
_bounds.last  = INVALID_LONG;
	} else {
		HFSM2_ASSERT(_bounds.first == INVALID_LONG);
		HFSM2_ASSERT(_bounds.last  == INVALID_LONG);
	}
}

template <typename TArgs>
HFSM2_CONSTEXPR(14)
void
PlanT<TArgs>::clearStatuses() noexcept {
TasksBits bitsToClear;
	bitsToClear.set();

const StateID begin = _registry.regionHeads[_regionId];

const StateID end   = _registry.regionHeads[_regionId] +
	_registry.regionSizes[_regionId];

for (StateID i = begin; i < end; ++i)
		bitsToClear.clear(i);

_planData.tasksSuccesses &= bitsToClear;
_planData.tasksFailures  &= bitsToClear;

_planData.headStatuses[_regionId].clear();
_planData. subStatuses[_regionId].clear();
}

template <typename TArgs>
HFSM2_CONSTEXPR(14)
PlanT<TArgs>::operator bool() const noexcept {
	HFSM2_ASSERT(_bounds.first < TASK_CAPACITY &&
				 _bounds.last  < TASK_CAPACITY ||
				 _bounds.last == INVALID_LONG);

return _bounds.first < TASK_CAPACITY;
}

template <typename TArgs>
HFSM2_CONSTEXPR(14)
void
PlanT<TArgs>::clear() noexcept {
	clearTasks();
	clearStatuses();
}

template <typename TArgs>
HFSM2_CONSTEXPR(14)
void
PlanT<TArgs>::remove(const Long index) noexcept {
	HFSM2_ASSERT(_planData.planExists.get(_regionId));
	HFSM2_ASSERT(_bounds.first < TaskLinks::CAPACITY);
	HFSM2_ASSERT(_bounds.last  < TaskLinks::CAPACITY);

	HFSM2_ASSERT(index < TaskLinks::CAPACITY);

TaskLink& link = _planData.taskLinks[index];

	if (link.prev < TaskLinks::CAPACITY) {
TaskLink& prev = _planData.taskLinks[link.prev];
prev.next = link.next;
	} else {
		HFSM2_ASSERT(_bounds.first == index);
_bounds.first = link.next;
	}

	if (link.next < TaskLinks::CAPACITY) {
TaskLink& next = _planData.taskLinks[link.next];
next.prev = link.prev;
	} else {
		HFSM2_ASSERT(_bounds.last == index);
_bounds.last = link.prev;
	}

link.prev = INVALID_LONG;
link.next = INVALID_LONG;

	_planData.tasks.remove(index);
}

}
}

#endif

#if HFSM2_PLANS_AVAILABLE()

namespace hfsm2 {
namespace detail {

template <typename TArgs>
class PayloadPlanT;

template <
	typename TConfig
  , typename TStateList
  , typename TRegionList
  , Long NCompoCount
  , Long NOrthoCount
  , Long NOrthoUnits
  , typename TReactOrder
  HFSM2_IF_SERIALIZATION(, Long NSerialBits)
  , Long NTaskCapacity
  , typename TPayload
>
class PayloadPlanT<
		  ArgsT<
			  TConfig
			, TStateList
			, TRegionList
			, NCompoCount
			, NOrthoCount
			, NOrthoUnits
			, TReactOrder
			HFSM2_IF_SERIALIZATION(, NSerialBits)
			, NTaskCapacity
			, TPayload
		  >
	  > final
	: public PlanT<
				 ArgsT<
					 TConfig
				   , TStateList
				   , TRegionList
				   , NCompoCount
				   , NOrthoCount
				   , NOrthoUnits
				   , TReactOrder
				   HFSM2_IF_SERIALIZATION(, NSerialBits)
				   , NTaskCapacity
				   , TPayload
				 >
			 >
{
	template <typename>
	friend class PlanControlT;

	template <typename>
	friend class FullControlT;

	template <typename>
	friend class GuardControlT;

	template <typename, typename>
	friend class R_;

	using Args = ArgsT<
					 TConfig
				   , TStateList
				   , TRegionList
				   , NCompoCount
				   , NOrthoCount
				   , NOrthoUnits
				   , TReactOrder
				   HFSM2_IF_SERIALIZATION(, NSerialBits)
				   , NTaskCapacity
				   , TPayload
				 >;

	using Payload		= typename Args::Payload;

	static constexpr Long  TASK_CAPACITY	= Args::TASK_CAPACITY;

	using PlanBase		= PlanT<Args>;

	using PlanBase::PlanBase;

	using PlanBase::linkTask;

	HFSM2_CONSTEXPR(14)	bool  append(const StateID origin,
									 const StateID destination,
									 const TransitionType type,
									 const Payload& payload)			noexcept;

public:

	/// @brief Append a task to transition from `origin` to `destination` if `origin` completes with `success()`
	///   (if transitioning into a region, acts depending on the region type)
	/// @param `origin` Origin state identifier
	/// @param `destination` Destination state identifier
	/// @param `payload` Payload
	/// @return Seccess if FSM total number of tasks is below task capacity
	/// @note use `Config::TaskCapacityN<>` to increase task capacity if necessary
	HFSM2_CONSTEXPR(14)	bool changeWith   (const StateID origin,
										   const StateID destination,
										   const Payload& payload)		noexcept	{ return append(origin								 , destination								 , TransitionType::CHANGE   ,	   payload );	}

	/// @brief Append a task to transition from `origin` to `destination` if `origin` completes with `success()`
	///   (if transitioning into a region, acts depending on the region type)
	/// @tparam `TOrigin` Origin state type
	/// @param `destination` Destination state identifier
	/// @param `payload` Payload
	/// @return Seccess if FSM total number of tasks is below task capacity
	/// @note use `Config::TaskCapacityN<>` to increase task capacity if necessary
	template <typename TOrigin>
	HFSM2_CONSTEXPR(14)	bool changeWith   (const StateID destination,
										   const Payload& payload)		noexcept	{ return append(PlanBase::template stateId<TOrigin>(), destination								 , TransitionType::CHANGE   ,	   payload );	}

	/// @brief Prepend a task to transition from `origin` to `destination` if `origin` completes with `success()`
	///   (if transitioning into a region, acts depending on the region type)
	/// @tparam `TOrigin` Origin state type
	/// @tparam `TDestination` Destination state type
	/// @param `payload` Payload
	/// @return Seccess if FSM total number of tasks is below task capacity
	/// @note use `Config::TaskCapacityN<>` to increase task capacity if necessary
	template <typename TOrigin, typename TDestination>
	HFSM2_CONSTEXPR(14)	bool changeWith   (const Payload& payload)		noexcept	{ return append(PlanBase::template stateId<TOrigin>(), PlanBase::template stateId<TDestination>(), TransitionType::CHANGE   ,	   payload );	}

	/// @brief Append a task to transition from `origin` to `destination` if `origin` completes with `success()`
	///   (if transitioning into a region, activates the initial state)
	/// @param `origin` Origin state identifier
	/// @param `destination` Destination state identifier
	/// @param `payload` Payload
	/// @return Seccess if FSM total number of tasks is below task capacity
	/// @note use `Config::TaskCapacityN<>` to increase task capacity if necessary
	HFSM2_CONSTEXPR(14)	bool restartWith  (const StateID origin,
										   const StateID destination,
										   const Payload& payload)		noexcept	{ return append(origin								 , destination								 , TransitionType::RESTART  ,	   payload );	}

	/// @brief Append a task to transition from `origin` to `destination` if `origin` completes with `success()`
	///   (if transitioning into a region, activates the initial state)
	/// @tparam `TOrigin` Origin state type
	/// @param `destination` Destination state identifier
	/// @param `payload` Payload
	/// @return Seccess if FSM total number of tasks is below task capacity
	/// @note use `Config::TaskCapacityN<>` to increase task capacity if necessary
	template <typename TOrigin>
	HFSM2_CONSTEXPR(14)	bool restartWith  (const StateID destination,
										   const Payload& payload)		noexcept	{ return append(PlanBase::template stateId<TOrigin>(), destination								 , TransitionType::RESTART  ,	   payload );	}

	/// @brief Prepend a task to transition from `origin` to `destination` if `origin` completes with `success()`
	///   (if transitioning into a region, activates the initial state)
	/// @tparam `TOrigin` Origin state type
	/// @tparam `TDestination` Destination state type
	/// @param `payload` Payload
	/// @return Seccess if FSM total number of tasks is below task capacity
	/// @note use `Config::TaskCapacityN<>` to increase task capacity if necessary
	template <typename TOrigin, typename TDestination>
	HFSM2_CONSTEXPR(14)	bool restartWith  (const Payload& payload)		noexcept	{ return append(PlanBase::template stateId<TOrigin>(), PlanBase::template stateId<TDestination>(), TransitionType::RESTART  ,	   payload );	}

	/// @brief Append a task to transition from `origin` to `destination` if `origin` completes with `success()`
	///   (if transitioning into a region, activates the state that was active previously)
	/// @param `origin` Origin state identifier
	/// @param `destination` Destination state identifier
	/// @param `payload` Payload
	/// @return Seccess if FSM total number of tasks is below task capacity
	/// @note use `Config::TaskCapacityN<>` to increase task capacity if necessary
	HFSM2_CONSTEXPR(14)	bool resumeWith   (const StateID origin,
										   const StateID destination,
										   const Payload& payload)		noexcept	{ return append(origin								 , destination								 , TransitionType::RESUME   ,	   payload );	}

	/// @brief Append a task to transition from `origin` to `destination` if `origin` completes with `success()`
	///   (if transitioning into a region, activates the state that was active previously)
	/// @tparam `TOrigin` Origin state type
	/// @param `destination` Destination state identifier
	/// @param `payload` Payload
	/// @return Seccess if FSM total number of tasks is below task capacity
	/// @note use `Config::TaskCapacityN<>` to increase task capacity if necessary
	template <typename TOrigin>
	HFSM2_CONSTEXPR(14)	bool resumeWith   (const StateID destination,
										   const Payload& payload)		noexcept	{ return append(PlanBase::template stateId<TOrigin>(), destination								 , TransitionType::RESUME   ,	   payload );	}

	/// @brief Prepend a task to transition from `origin` to `destination` if `origin` completes with `success()`
	///   (if transitioning into a region, activates the state that was active previously)
	/// @tparam `TOrigin` Origin state type
	/// @tparam `TDestination` Destination state type
	/// @param `payload` Payload
	/// @return Seccess if FSM total number of tasks is below task capacity
	/// @note use `Config::TaskCapacityN<>` to increase task capacity if necessary
	template <typename TOrigin, typename TDestination>
	HFSM2_CONSTEXPR(14)	bool resumeWith   (const Payload& payload)		noexcept	{ return append(PlanBase::template stateId<TOrigin>(), PlanBase::template stateId<TDestination>(), TransitionType::RESUME   ,	   payload );	}

	/// @brief Append a task to transition from `origin` to `destination` if `origin` completes with `success()`
	///   (if transitioning into a region, activates the sub-state by index returned by the region's `select()` method)
	/// @param `origin` Origin state identifier
	/// @param `destination` Destination state identifier
	/// @param `payload` Payload
	/// @return Seccess if FSM total number of tasks is below task capacity
	/// @note use `Config::TaskCapacityN<>` to increase task capacity if necessary
	HFSM2_CONSTEXPR(14)	bool selectWith   (const StateID origin,
										   const StateID destination,
										   const Payload& payload)		noexcept	{ return append(origin								 , destination								 , TransitionType::SELECT   ,	   payload );	}

	/// @brief Append a task to transition from `origin` to `destination` if `origin` completes with `success()`
	///   (if transitioning into a region, activates the sub-state by index returned by the region's `select()` method)
	/// @tparam `TOrigin` Origin state type
	/// @param `destination` Destination state identifier
	/// @param `payload` Payload
	/// @return Seccess if FSM total number of tasks is below task capacity
	/// @note use `Config::TaskCapacityN<>` to increase task capacity if necessary
	template <typename TOrigin>
	HFSM2_CONSTEXPR(14)	bool selectWith   (const StateID destination,
										   const Payload& payload)		noexcept	{ return append(PlanBase::template stateId<TOrigin>(), destination								 , TransitionType::SELECT   ,	   payload );	}

	/// @brief Prepend a task to transition from `origin` to `destination` if `origin` completes with `success()`
	///   (if transitioning into a region, activates the sub-state by index returned by the region's `select()` method)
	/// @tparam `TOrigin` Origin state type
	/// @tparam `TDestination` Destination state type
	/// @param `payload` Payload
	/// @return Seccess if FSM total number of tasks is below task capacity
	/// @note use `Config::TaskCapacityN<>` to increase task capacity if necessary
	template <typename TOrigin, typename TDestination>
	HFSM2_CONSTEXPR(14)	bool selectWith   (const Payload& payload)		noexcept	{ return append(PlanBase::template stateId<TOrigin>(), PlanBase::template stateId<TDestination>(), TransitionType::SELECT   ,	   payload );	}

#if HFSM2_UTILITY_THEORY_AVAILABLE()

	/// @brief Append a task to transition from `origin` to `destination` if `origin` completes with `success()`
	///   (if transitioning into a region, activates the state with the highest `utility()`
	///   among those with the highest `rank()`)
	/// @param `origin` Origin state identifier
	/// @param `destination` Destination state identifier
	/// @param `payload` Payload
	/// @return Seccess if FSM total number of tasks is below task capacity
	/// @note use `Config::TaskCapacityN<>` to increase task capacity if necessary
	/// @see `HFSM2_ENABLE_UTILITY_THEORY`
	HFSM2_CONSTEXPR(14)	bool utilizeWith  (const StateID origin,
										   const StateID destination,
										   const Payload& payload)		noexcept	{ return append(origin								 , destination								 , TransitionType::UTILIZE  ,	   payload );	}

	/// @brief Append a task to transition from `origin` to `destination` if `origin` completes with `success()`
	///   (if transitioning into a region, activates the state with the highest `utility()`
	///   among those with the highest `rank()`)
	/// @tparam `TOrigin` Origin state type
	/// @param `destination` Destination state identifier
	/// @param `payload` Payload
	/// @return Seccess if FSM total number of tasks is below task capacity
	/// @note use `Config::TaskCapacityN<>` to increase task capacity if necessary
	/// @see `HFSM2_ENABLE_UTILITY_THEORY`
	template <typename TOrigin>
	HFSM2_CONSTEXPR(14)	bool utilizeWith  (const StateID destination,
										   const Payload& payload)		noexcept	{ return append(PlanBase::template stateId<TOrigin>(), destination								 , TransitionType::UTILIZE  ,	   payload );	}

	/// @brief Prepend a task to transition from `origin` to `destination` if `origin` completes with `success()`
	///   (if transitioning into a region, activates the state with the highest `utility()`
	///   among those with the highest `rank()`)
	/// @tparam `TOrigin` Origin state type
	/// @tparam `TDestination` Destination state type
	/// @param `payload` Payload
	/// @return Seccess if FSM total number of tasks is below task capacity
	/// @note use `Config::TaskCapacityN<>` to increase task capacity if necessary
	/// @see `HFSM2_ENABLE_UTILITY_THEORY`
	template <typename TOrigin, typename TDestination>
	HFSM2_CONSTEXPR(14)	bool utilizeWith  (const Payload& payload)		noexcept	{ return append(PlanBase::template stateId<TOrigin>(), PlanBase::template stateId<TDestination>(), TransitionType::UTILIZE  ,	   payload );	}

	/// @brief Append a task to transition from `origin` to `destination` if `origin` completes with `success()`
	///   (if transitioning into a region, uses weighted random to activate the state proportional to `utility()`
	///   among those with the highest `rank()`)
	/// @param `origin` Origin state identifier
	/// @param `destination` Destination state identifier
	/// @param `payload` Payload
	/// @return Seccess if FSM total number of tasks is below task capacity
	/// @note use `Config::TaskCapacityN<>` to increase task capacity if necessary
	/// @see `HFSM2_ENABLE_UTILITY_THEORY`
	HFSM2_CONSTEXPR(14)	bool randomizeWith(const StateID origin,
										   const StateID destination,
										   const Payload& payload)		noexcept	{ return append(origin								 , destination								 , TransitionType::RANDOMIZE,	   payload );	}

	/// @brief Append a task to transition from `origin` to `destination` if `origin` completes with `success()`
	///   (if transitioning into a region, uses weighted random to activate the state proportional to `utility()`
	///   among those with the highest `rank()`)
	/// @tparam `TOrigin` Origin state type
	/// @param `destination` Destination state identifier
	/// @param `payload` Payload
	/// @return Seccess if FSM total number of tasks is below task capacity
	/// @note use `Config::TaskCapacityN<>` to increase task capacity if necessary
	/// @see `HFSM2_ENABLE_UTILITY_THEORY`
	template <typename TOrigin>
	HFSM2_CONSTEXPR(14)	bool randomizeWith(const StateID destination,
										   const Payload& payload)		noexcept	{ return append(PlanBase::template stateId<TOrigin>(), destination								 , TransitionType::RANDOMIZE,	   payload );	}

	/// @brief Prepend a task to transition from `origin` to `destination` if `origin` completes with `success()`
	///   (if transitioning into a region, uses weighted random to activate the state proportional to `utility()`
	///   among those with the highest `rank()`)
	/// @tparam `TOrigin` Origin state type
	/// @tparam `TDestination` Destination state type
	/// @param `payload` Payload
	/// @return Seccess if FSM total number of tasks is below task capacity
	/// @note use `Config::TaskCapacityN<>` to increase task capacity if necessary
	/// @see `HFSM2_ENABLE_UTILITY_THEORY`
	template <typename TOrigin, typename TDestination>
	HFSM2_CONSTEXPR(14)	bool randomizeWith(const Payload& payload)		noexcept	{ return append(PlanBase::template stateId<TOrigin>(), PlanBase::template stateId<TDestination>(), TransitionType::RANDOMIZE,	   payload );	}

#endif

	/// @brief Append a task to schedule a transition to `destination` if `origin` completes with `success()`
	/// @param `origin` Origin state identifier
	/// @param `destination` Destination state identifier
	/// @param `payload` Payload
	/// @return Seccess if FSM total number of tasks is below task capacity
	/// @note use `Config::TaskCapacityN<>` to increase task capacity if necessary
	HFSM2_CONSTEXPR(14)	bool scheduleWith (const StateID origin,
										   const StateID destination,
										   const Payload& payload)		noexcept	{ return append(origin								 , destination								 , TransitionType::SCHEDULE ,	   payload );	}

	/// @brief Append a task to schedule a transition to `destination` if `origin` completes with `success()`
	/// @tparam `TOrigin` Origin state type
	/// @param `destination` Destination state identifier
	/// @param `payload` Payload
	/// @return Seccess if FSM total number of tasks is below task capacity
	/// @note use `Config::TaskCapacityN<>` to increase task capacity if necessary
	template <typename TOrigin>
	HFSM2_CONSTEXPR(14)	bool scheduleWith (const StateID destination,
										   const Payload& payload)		noexcept	{ return append(PlanBase::template stateId<TOrigin>(), destination								 , TransitionType::SCHEDULE ,	   payload );	}

	/// @brief Prepend a task to schedule a transition to `destination` if `origin` completes with `success()`
	/// @tparam `TOrigin` Origin state type
	/// @tparam `TDestination` Destination state type
	/// @param `payload` Payload
	/// @return Seccess if FSM total number of tasks is below task capacity
	/// @note use `Config::TaskCapacityN<>` to increase task capacity if necessary
	template <typename TOrigin, typename TDestination>
	HFSM2_CONSTEXPR(14)	bool scheduleWith (const Payload& payload)		noexcept	{ return append(PlanBase::template stateId<TOrigin>(), PlanBase::template stateId<TDestination>(), TransitionType::SCHEDULE ,	   payload );	}

private:
	using PlanBase::_planData;
using PlanBase::_regionId;
};

template <
	typename TConfig
  , typename TStateList
  , typename TRegionList
  , Long NCompoCount
  , Long NOrthoCount
  , Long NOrthoUnits
  , typename TReactOrder
  HFSM2_IF_SERIALIZATION(, Long NSerialBits)
  , Long NTaskCapacity
>
class PayloadPlanT<
		  ArgsT<
			  TConfig
			, TStateList
			, TRegionList
			, NCompoCount
			, NOrthoCount
			, NOrthoUnits
			, TReactOrder
			HFSM2_IF_SERIALIZATION(, NSerialBits)
			, NTaskCapacity
			, void
		  >
	  > final
	: public PlanT<
				 ArgsT<
					 TConfig
				   , TStateList
				   , TRegionList
				   , NCompoCount
				   , NOrthoCount
				   , NOrthoUnits
				   , TReactOrder
				   HFSM2_IF_SERIALIZATION(, NSerialBits)
				   , NTaskCapacity
				   , void
				 >
			 >
{
	template <typename, typename>
	friend class R_;

	template <typename>
	friend class PlanControlT;

	template <typename>
	friend class FullControlT;

	template <typename>
	friend class GuardControlT;

	using Args = ArgsT<
	TConfig
	, TStateList
	, TRegionList
	, NCompoCount
	, NOrthoCount
	, NOrthoUnits
	, TReactOrder
				   HFSM2_IF_SERIALIZATION(, NSerialBits)
				   , NTaskCapacity
				   , void
				 >;

	using PlanBase = PlanT<Args>;

using PlanBase::PlanBase;
};

}
}

#endif

#if HFSM2_PLANS_AVAILABLE()

namespace hfsm2 {
namespace detail {

template <typename TG_, typename TSL_, typename TRL_, Long NCC_, Long NOC_, Long NOU_, typename TRO_ HFSM2_IF_SERIALIZATION(, Long NSB_), Long NTC_, typename TTP_>
HFSM2_CONSTEXPR(14)
bool
PayloadPlanT<ArgsT<TG_, TSL_, TRL_, NCC_, NOC_, NOU_, TRO_ HFSM2_IF_SERIALIZATION(, NSB_), NTC_, TTP_>>:: append(const StateID origin,
																												 const StateID destination,
																												 const TransitionType transitionType,
																												 const Payload& payload) noexcept
{
	if (_planData.tasks.count() < TASK_CAPACITY) {
		_planData.planExists.set(_regionId);

		return linkTask(_planData.tasks.emplace(origin, destination, transitionType, payload));
	} else
		return false;
}

}
}

#endif

namespace hfsm2 {
	namespace detail {

		template <typename TArgs>
		struct CoreT {
			using Context			= typename TArgs::Context;
			using PureContext		= typename TArgs::PureContext;

			using Registry			= RegistryT<TArgs>;

			using Payload			= typename TArgs::Payload;
			using Transition		= TransitionT<Payload>;
			using TransitionSet		= DynamicArrayT<Transition, TArgs::COMPO_COUNT>;
			using TransitionSets	= DynamicArrayT<Transition, TArgs::COMPO_COUNT * TArgs::SUBSTITUTION_LIMIT>;

#if HFSM2_PLANS_AVAILABLE()
			using PlanData			= PlanDataT<TArgs>;
#endif

#if HFSM2_TRANSITION_HISTORY_AVAILABLE()
			using TransitionTargets	= StaticArrayT<Short, TArgs::STATE_COUNT>;
#endif

#if HFSM2_UTILITY_THEORY_AVAILABLE()
			using RNG				= typename TArgs::RNG;
#endif

#if HFSM2_LOG_INTERFACE_AVAILABLE()
			using Logger			= typename TArgs::Logger;
#endif

			HFSM2_CONSTEXPR(14)	explicit CoreT(Context& context_
			HFSM2_IF_UTILITY_THEORY(, RNG& rng_)
			HFSM2_IF_LOG_INTERFACE(, Logger* const logger_ = nullptr))		noexcept;

			HFSM2_CONSTEXPR(14)	explicit CoreT(PureContext&& context_
			HFSM2_IF_UTILITY_THEORY(, RNG& rng_)
			HFSM2_IF_LOG_INTERFACE(, Logger* const logger_ = nullptr))		noexcept;

			HFSM2_CONSTEXPR(14) CoreT(const CoreT&  other)													noexcept;
			HFSM2_CONSTEXPR(14) CoreT(		CoreT&& other)													noexcept;

			Context context;
			Registry registry;
			TransitionSet requests;
			HFSM2_IF_PLANS(PlanData planData);
			HFSM2_IF_TRANSITION_HISTORY(TransitionTargets transitionTargets);
			HFSM2_IF_TRANSITION_HISTORY(TransitionSets previousTransitions);
			HFSM2_IF_UTILITY_THEORY(RNG& rng);
			HFSM2_IF_LOG_INTERFACE(Logger* logger);
		};

	}
}

namespace hfsm2 {
	namespace detail {

		template <typename TArgs>
		HFSM2_CONSTEXPR(14)
		CoreT<TArgs>::CoreT(Context& context_
		HFSM2_IF_UTILITY_THEORY(, RNG& rng_)
		HFSM2_IF_LOG_INTERFACE(, Logger* const logger_)) noexcept
	: context{context_}
	HFSM2_IF_UTILITY_THEORY(, rng{rng_})
	HFSM2_IF_LOG_INTERFACE(, logger{logger_})
{}

template <typename TArgs>
HFSM2_CONSTEXPR(14)
CoreT<TArgs>::CoreT(PureContext&& context_
				  HFSM2_IF_UTILITY_THEORY(, RNG& rng_)
				  HFSM2_IF_LOG_INTERFACE(, Logger* const logger_)) noexcept
	: context{move(context_)}
HFSM2_IF_UTILITY_THEORY(, rng	{rng_	})
HFSM2_IF_LOG_INTERFACE (, logger{logger_})
{}

template <typename TArgs>
HFSM2_CONSTEXPR(14)
CoreT<TArgs>::CoreT(const CoreT& other) noexcept
	: context {other.context }
	, registry{other.registry}
	, requests{other.requests}
HFSM2_IF_PLANS			   (, planData			 {other.planData		   })
HFSM2_IF_TRANSITION_HISTORY(, transitionTargets  {other.transitionTargets  })
HFSM2_IF_TRANSITION_HISTORY(, previousTransitions{other.previousTransitions})
HFSM2_IF_UTILITY_THEORY	   (, rng				 {other.rng				   })
HFSM2_IF_LOG_INTERFACE	   (, logger			 {other.logger			   })
{}

template <typename TArgs>
HFSM2_CONSTEXPR(14)
CoreT<TArgs>::CoreT(CoreT&& other) noexcept
	: context {move(other.context )}
	, registry{move(other.registry)}
	, requests{move(other.requests)}
HFSM2_IF_PLANS			   (, planData			 {move(other.planData			)})
HFSM2_IF_TRANSITION_HISTORY(, transitionTargets  {move(other.transitionTargets	)})
HFSM2_IF_TRANSITION_HISTORY(, previousTransitions{move(other.previousTransitions)})
HFSM2_IF_UTILITY_THEORY	   (, rng				 {move(other.rng				)})
HFSM2_IF_LOG_INTERFACE	   (, logger			 {move(other.logger				)})
{}

}
}

namespace hfsm2 {
	namespace detail {

		template <typename TArgs>
		class ConstControlT {
			template <typename, typename, typename>
			friend struct S_;

			template <typename, typename, Strategy, typename, typename...>
			friend struct C_;

			template <typename, typename, typename, typename...>
			friend struct O_;

			template <typename, typename>
			friend class R_;

			template <typename, typename>
			friend struct QueryWrapperT;

			protected:
			using Context			= typename TArgs::Context;

			using StateList			= typename TArgs::StateList;
			using RegionList		= typename TArgs::RegionList;

			using Core				= CoreT	   <TArgs>;
			using Registry			= RegistryT<TArgs>;

			using Payload			= typename TArgs::Payload;
			using Transition		= TransitionT<Payload>;
			using TransitionSet		= DynamicArrayT<Transition, TArgs::COMPO_COUNT>;
			using TransitionSets	= DynamicArrayT<Transition, TArgs::COMPO_COUNT * TArgs::SUBSTITUTION_LIMIT>;

#if HFSM2_TRANSITION_HISTORY_AVAILABLE()
			using TransitionTargets	= StaticArrayT<Short, TArgs::STATE_COUNT>;
#endif

#if HFSM2_UTILITY_THEORY_AVAILABLE()
			using RNG				= typename TArgs::RNG;
#endif

#if HFSM2_PLANS_AVAILABLE()
			using PlanData			= PlanDataT<TArgs>;
#endif

#if HFSM2_LOG_INTERFACE_AVAILABLE()
			using Logger			= typename TArgs::Logger;
#endif

			struct Origin final {
			HFSM2_CONSTEXPR(14)	 Origin(ConstControlT& control_,
			const StateID stateId_)					noexcept;

			HFSM2_CONSTEXPR(20)	~Origin()										noexcept;

			ConstControlT& control;
			const StateID prevId;
		};

		struct Region {
			HFSM2_CONSTEXPR(14)	 Region(ConstControlT& control,
			const RegionID regionId_)				noexcept;

			HFSM2_CONSTEXPR(20)	~Region()										noexcept;

			ConstControlT& control;
			const RegionID prevId;
		};

		HFSM2_CONSTEXPR(11)	ConstControlT(const Core& core)						noexcept
	: _core{core}
{}

	HFSM2_CONSTEXPR(14)	void   setRegion(const RegionID regionId_)			noexcept;
	HFSM2_CONSTEXPR(14)	void resetRegion(const RegionID regionId_)			noexcept;

#if HFSM2_TRANSITION_HISTORY_AVAILABLE()
	HFSM2_CONSTEXPR(14)	void pinLastTransition(const StateID stateId_,
											   const Short index)			noexcept;
#endif

public:

#if HFSM2_PLANS_AVAILABLE()
	using CPlan				= CPlanT<TArgs>;
#endif

	/// @brief Get current state's identifier
	/// @return Numeric state identifier
	HFSM2_CONSTEXPR(11) StateID  stateId()							  const noexcept	{ return _originId;												}

	/// @brief Get state identifier for a state type
	/// @tparam `TState` State type
	/// @return Numeric state identifier
	template <typename TState>
	static
	HFSM2_CONSTEXPR(11) StateID  stateId()									noexcept	{ return					   index<StateList , TState>() ;	}

	/// @brief Get region identifier for a region type
	/// @tparam `TState` Region head state type
	/// @return Numeric region identifier
	template <typename TState>
	static
	HFSM2_CONSTEXPR(11) RegionID regionId()									noexcept	{ return static_cast<RegionID>(index<RegionList, TState>());	}

	/// @brief Access FSM context (data shared between states and/or data interface between FSM and external code)
	/// @return context
	/// @see Control::context()
	HFSM2_CONSTEXPR(11)	const Context& _()							  const noexcept	{ return _core.context;											}

	/// @brief Access FSM context (data shared between states and/or data interface between FSM and external code)
	/// @return context
	/// @see Control::_()
	HFSM2_CONSTEXPR(11)	const Context& context()					  const noexcept	{ return _core.context;											}

	/// @brief Stops processing of the current query down the hierarchy
	/// @see Config::BottomUpReactions
	HFSM2_CONSTEXPR(14)	void consumeQuery()									noexcept	{ _consumed = true;												}

	/// @brief Inspect current transition requests
	/// @return Array of transition requests
	HFSM2_CONSTEXPR(11)	const TransitionSet& requests()				  const noexcept	{ return _core.requests;										}

	/// @brief Get active sub-state's index for the current region
	/// @return Region's active sub-state index
	HFSM2_CONSTEXPR(14)	Prong activeSubState()						  const noexcept	{ return _core.registry.activeSubState(_originId);				}

	/// @brief Get region's active sub-state's index
	/// @param `stateId` Region's head state identifier
	/// @return Region's active sub-state index
	HFSM2_CONSTEXPR(14)	Prong activeSubState(const StateID stateId_)  const noexcept	{ return _core.registry.activeSubState(stateId_);				}

	/// @brief Get region's active sub-state's index
	/// @tparam `TState` Region's head state type
	/// @return Region's active sub-state index
	template <typename TState>
	HFSM2_CONSTEXPR(14)	Prong activeSubState()						  const noexcept	{ return _core.registry.activeSubState(stateId<TState>());		}

	/// @brief Check if a state is active
	/// @param `stateId` State identifier
	/// @return State active status
	HFSM2_CONSTEXPR(11)	bool isActive   (const StateID stateId_)	  const noexcept	{ return _core.registry.isActive(stateId_);						}

	/// @brief Check if a state is active
	/// @tparam `TState` State type
	/// @return State active status
	template <typename TState>
	HFSM2_CONSTEXPR(11)	bool isActive	()							  const noexcept	{ return isActive(stateId<TState>());							}

	/// @brief Check if a state is resumable (activated then deactivated previously)
	/// @param `stateId` State identifier
	/// @return State resumable status
	HFSM2_CONSTEXPR(11)	bool isResumable(const StateID stateId_)	  const noexcept	{ return _core.registry.isResumable(stateId_);					}

	/// @brief Check if a state is resumable (activated then deactivated previously)
	/// @tparam `TState` State type
	/// @return State resumable status
	template <typename TState>
	HFSM2_CONSTEXPR(11)	bool isResumable()							  const noexcept	{ return isResumable(stateId<TState>());						}

	/// @brief Check if a state is scheduled to activate on the next transition to parent region
	/// @param `stateId` State identifier
	/// @return State scheduled status
	HFSM2_CONSTEXPR(11)	bool isScheduled(const StateID stateId_)	  const noexcept	{ return isResumable(stateId_);									}

	/// @brief Check if a state is scheduled to activate on the next transition to parent region
	/// @tparam `TState` State type
	/// @return State scheduled status
	template <typename TState>
	HFSM2_CONSTEXPR(11)	bool isScheduled()							  const noexcept	{ return isResumable(stateId<TState>());						}

#if HFSM2_PLANS_AVAILABLE()

	/// @brief Access read-only plan for the current region
	/// @return Plan for the current region
	/// @see `HFSM2_ENABLE_PLANS`
	HFSM2_CONSTEXPR(11)	CPlan plan()								  const noexcept	{ return CPlan{_core.registry, _core.planData, _regionId};						}

	/// @brief Access read-only plan for a region
	/// @param `regionId` Region identifier
	/// @return Read-only plan for the region
	/// @see `HFSM2_ENABLE_PLANS`
	HFSM2_CONSTEXPR(14)	CPlan plan(const RegionID regionId_)		  const noexcept	{ return CPlan{_core.registry, _core.planData, regionId_};						}

	/// @brief Access read-only plan for a region
	/// @tparam `TRegion` Region head state type
	/// @return Read-only Plan for the region
	/// @see `HFSM2_ENABLE_PLANS`
	template <typename TRegion>
	HFSM2_CONSTEXPR(14)	CPlan plan()								  const noexcept	{ return CPlan{_core.registry, _core.planData, regionId<TRegion>()};			}

#endif

#if HFSM2_TRANSITION_HISTORY_AVAILABLE()

	/// @brief Get transitions processed during last `update()`, `react()` or `replayTransitions()`
	/// @return Array of last transition requests
	/// @see `HFSM2_ENABLE_TRANSITION_HISTORY`
	HFSM2_CONSTEXPR(11)	const TransitionSets& previousTransitions()					  const noexcept	{ return _core.previousTransitions;				}

	/// @brief Get the last transition that caused the state to be activated
	/// @param `stateId` State identifier
	/// @return Pointer to the last transition that activated the state
	/// @see `HFSM2_ENABLE_TRANSITION_HISTORY`
	HFSM2_CONSTEXPR(14)	const Transition* lastTransitionTo(const StateID stateId_)	  const noexcept;

	/// @brief Get the last transition that caused the state to be activated
	/// @tparam `TState` State type
	/// @return Pointer to the last transition that activated the state
	/// @see `HFSM2_ENABLE_TRANSITION_HISTORY`
	template <typename TState>
	HFSM2_CONSTEXPR(11)	const Transition* lastTransitionTo()						  const noexcept	{ return lastTransitionTo(stateId<TState>());	}

	/// @brief Get the last transition that caused the current state to be activated
	/// @return Pointer to the last transition that activated the current state
	/// @see `HFSM2_ENABLE_TRANSITION_HISTORY`
	HFSM2_CONSTEXPR(14)	const Transition* lastTransition()							  const noexcept;

#endif

protected:
const Core& _core;
StateID _originId = INVALID_STATE_ID;
RegionID _regionId = 0;
bool _consumed = false;
};

}
}

namespace hfsm2 {
	namespace detail {

		template <typename TArgs>
		HFSM2_CONSTEXPR(14)
		ConstControlT<TArgs>::Origin::Origin(ConstControlT& control_,
		const StateID stateId_) noexcept
	: control{control_}
, prevId{control._originId}
{
	HFSM2_ASSERT(stateId_ < StateList::SIZE);
control._originId = stateId_;
}

template <typename TArgs>
HFSM2_CONSTEXPR(20)
ConstControlT<TArgs>::Origin::~Origin() noexcept {
control._originId = prevId;
}

template <typename TArgs>
HFSM2_CONSTEXPR(14)
ConstControlT<TArgs>::Region::Region(ConstControlT& control_,
									 const RegionID regionId_) noexcept
	: control{control_}
	, prevId{control._regionId}
{
	control.setRegion(regionId_);
}

template <typename TArgs>
HFSM2_CONSTEXPR(20)
ConstControlT<TArgs>::Region::~Region() noexcept {
	control.resetRegion(prevId);
}

template <typename TArgs>
HFSM2_CONSTEXPR(14)
void
ConstControlT<TArgs>::setRegion(const RegionID regionId_) noexcept {
	HFSM2_ASSERT(_regionId <= regionId_ && regionId_ < RegionList::SIZE);

_regionId = regionId_;
}

template <typename TArgs>
HFSM2_CONSTEXPR(14)
void
ConstControlT<TArgs>::resetRegion(const RegionID regionId_) noexcept {
	HFSM2_ASSERT(regionId_ <= _regionId && _regionId < RegionList::SIZE);

_regionId = regionId_;
}

}
}

namespace hfsm2 {
	namespace detail {

		template <typename TArgs>
		class ControlT {
			template <typename, typename, typename>
			friend struct S_;

			template <typename, typename, Strategy, typename, typename...>
			friend struct C_;

			template <typename, typename, typename, typename...>
			friend struct O_;

			template <typename, typename>
			friend class R_;

			protected:
			using Context			= typename TArgs::Context;

			using StateList			= typename TArgs::StateList;
			using RegionList		= typename TArgs::RegionList;

			using Core				= CoreT	   <TArgs>;
			using Registry			= RegistryT<TArgs>;

			using Payload			= typename TArgs::Payload;
			using Transition		= TransitionT<Payload>;
			using TransitionSet		= DynamicArrayT<Transition, TArgs::COMPO_COUNT>;
			using TransitionSets	= DynamicArrayT<Transition, TArgs::COMPO_COUNT * TArgs::SUBSTITUTION_LIMIT>;

#if HFSM2_TRANSITION_HISTORY_AVAILABLE()
			using TransitionTargets	= StaticArrayT<Short, TArgs::STATE_COUNT>;
#endif

#if HFSM2_UTILITY_THEORY_AVAILABLE()
			using RNG				= typename TArgs::RNG;
#endif

#if HFSM2_PLANS_AVAILABLE()
			using PlanData			= PlanDataT<TArgs>;
#endif

#if HFSM2_LOG_INTERFACE_AVAILABLE()
			using Logger			= typename TArgs::Logger;
#endif

			struct Origin final {
			HFSM2_CONSTEXPR(14)	 Origin(ControlT& control_,
			const StateID stateId_)					noexcept;

			HFSM2_CONSTEXPR(20)	~Origin()										noexcept;

			ControlT& control;
			const StateID prevId;
		};

		struct Region {
			HFSM2_CONSTEXPR(14)	 Region(ControlT& control,
			const RegionID regionId_)				noexcept;

			HFSM2_CONSTEXPR(20)	~Region()										noexcept;

			ControlT& control;
			const RegionID prevId;
		};

		HFSM2_CONSTEXPR(11)	ControlT(Core& core)								noexcept
	: _core{core}
{}

	HFSM2_CONSTEXPR(14)	void   setRegion(const RegionID regionId_)			noexcept;
	HFSM2_CONSTEXPR(14)	void resetRegion(const RegionID regionId_)			noexcept;

#if HFSM2_TRANSITION_HISTORY_AVAILABLE()
	HFSM2_CONSTEXPR(14)	void pinLastTransition(const StateID stateId_,
											   const Short index)			noexcept;
#endif

public:

#if HFSM2_PLANS_AVAILABLE()
	using CPlan				= CPlanT<TArgs>;
#endif

	/// @brief Get current state's identifier
	/// @return Numeric state identifier
	HFSM2_CONSTEXPR(11) StateID  stateId()							  const noexcept	{ return _originId;												}

	/// @brief Get state identifier for a state type
	/// @tparam `TState` State type
	/// @return Numeric state identifier
	template <typename TState>
	static
	HFSM2_CONSTEXPR(11) StateID  stateId()									noexcept	{ return					   index<StateList , TState>() ;	}

	/// @brief Get region identifier for a region type
	/// @tparam `TState` Region head state type
	/// @return Numeric region identifier
	template <typename TState>
	static
	HFSM2_CONSTEXPR(11) RegionID regionId()									noexcept	{ return static_cast<RegionID>(index<RegionList, TState>());	}

	/// @brief Access FSM context (data shared between states and/or data interface between FSM and external code)
	/// @return context
	/// @see `Control::context()`
	HFSM2_CONSTEXPR(14)		  Context& _()									noexcept	{ return _core.context;											}

	/// @brief Access FSM context (data shared between states and/or data interface between FSM and external code)
	/// @return context
	/// @see `Control::context()`
	HFSM2_CONSTEXPR(11)	const Context& _()							  const noexcept	{ return _core.context;											}

	/// @brief Access FSM context (data shared between states and/or data interface between FSM and external code)
	/// @return context
	/// @see `Control::_()`
	HFSM2_CONSTEXPR(14)		  Context& context()							noexcept	{ return _core.context;											}

	/// @brief Access FSM context (data shared between states and/or data interface between FSM and external code)
	/// @return context
	/// @see `Control::_()`
	HFSM2_CONSTEXPR(11)	const Context& context()					  const noexcept	{ return _core.context;											}

	/// @brief Inspect current transition requests
	/// @return Array of transition requests
	HFSM2_CONSTEXPR(11)	const TransitionSet& requests()				  const noexcept	{ return _core.requests;										}

	/// @brief Get active sub-state's index for the current region
	/// @return Region's active sub-state index
	HFSM2_CONSTEXPR(14)	Prong activeSubState()						  const noexcept	{ return _core.registry.activeSubState(_originId);				}

	/// @brief Get region's active sub-state's index
	/// @param `stateId` Region's head state ID
	/// @return Region's active sub-state index
	HFSM2_CONSTEXPR(14)	Prong activeSubState(const StateID stateId_)  const noexcept	{ return _core.registry.activeSubState(stateId_);				}

	/// @brief Get region's active sub-state's index
	/// @tparam `TState` Region's head state type
	/// @return Region's active sub-state index
	template <typename TState>
	HFSM2_CONSTEXPR(14)	Prong activeSubState()						  const noexcept	{ return _core.registry.activeSubState(stateId<TState>());		}

	/// @brief Check if a state is active
	/// @param `stateId` State identifier
	/// @return State active status
	HFSM2_CONSTEXPR(11)	bool isActive   (const StateID stateId_)	  const noexcept	{ return _core.registry.isActive(stateId_);						}

	/// @brief Check if a state is active
	/// @tparam `TState` State type
	/// @return State active status
	template <typename TState>
	HFSM2_CONSTEXPR(11)	bool isActive	()							  const noexcept	{ return isActive(stateId<TState>());							}

	/// @brief Check if a state is resumable (activated then deactivated previously)
	/// @param `stateId` State identifier
	/// @return State resumable status
	HFSM2_CONSTEXPR(11)	bool isResumable(const StateID stateId_)	  const noexcept	{ return _core.registry.isResumable(stateId_);					}

	/// @brief Check if a state is resumable (activated then deactivated previously)
	/// @tparam `TState` State type
	/// @return State resumable status
	template <typename TState>
	HFSM2_CONSTEXPR(11)	bool isResumable()							  const noexcept	{ return isResumable(stateId<TState>());						}

	/// @brief Check if a state is scheduled to activate on the next transition to parent region
	/// @param `stateId` State identifier
	/// @return State scheduled status
	HFSM2_CONSTEXPR(11)	bool isScheduled(const StateID stateId_)	  const noexcept	{ return isResumable(stateId_);									}

	/// @brief Check if a state is scheduled to activate on the next transition to parent region
	/// @tparam `TState` State type
	/// @return State scheduled status
	template <typename TState>
	HFSM2_CONSTEXPR(11)	bool isScheduled()							  const noexcept	{ return isResumable(stateId<TState>());						}

#if HFSM2_PLANS_AVAILABLE()

	/// @brief Access read-only plan for the current region
	/// @return Plan for the current region
	/// @see `HFSM2_ENABLE_PLANS`
	HFSM2_CONSTEXPR(11)	CPlan plan()								  const noexcept	{ return CPlan{_core.registry, _core.planData, _regionId};				}

	/// @brief Access read-only plan for a region
	/// @param `regionId` Region identifier
	/// @return Read-only plan for the region
	/// @see `HFSM2_ENABLE_PLANS`
	HFSM2_CONSTEXPR(14)	CPlan plan(const RegionID regionId_)		  const noexcept	{ return CPlan{_core.registry, _core.planData, regionId_};				}

	/// @brief Access read-only plan for a region
	/// @tparam `TRegion` Region head state type
	/// @return Read-only plan for the region
	/// @see `HFSM2_ENABLE_PLANS`
	template <typename TRegion>
	HFSM2_CONSTEXPR(14)	CPlan plan()										noexcept	{ return CPlan{_core.registry, _core.planData, regionId<TRegion>()};	}

	/// @brief Access read-only plan for a region
	/// @tparam `TRegion` Region head state type
	/// @return Read-only Plan for the region
	/// @see `HFSM2_ENABLE_PLANS`
	template <typename TRegion>
	HFSM2_CONSTEXPR(14)	CPlan plan()								  const noexcept	{ return CPlan{_core.registry, _core.planData, regionId<TRegion>()};	}

#endif

#if HFSM2_TRANSITION_HISTORY_AVAILABLE()

	/// @brief Get transitions processed during last `update()`, `react()` or `replayTransitions()`
	/// @return Array of last transition requests
	/// @see `HFSM2_ENABLE_TRANSITION_HISTORY`
	HFSM2_CONSTEXPR(11)	const TransitionSets& previousTransitions()					  const noexcept	{ return _core.previousTransitions;				}

	/// @brief Get the last transition that caused the state to be activated
	/// @param `stateId` State identifier
	/// @return Pointer to the last transition that activated the state
	/// @see `HFSM2_ENABLE_TRANSITION_HISTORY`
	HFSM2_CONSTEXPR(14)	const Transition* lastTransitionTo(const StateID stateId_)	  const noexcept;

	/// @brief Get the last transition that caused the state to be activated
	/// @tparam `TState` State type
	/// @return Pointer to the last transition that activated the state
	/// @see `HFSM2_ENABLE_TRANSITION_HISTORY`
	template <typename TState>
	HFSM2_CONSTEXPR(11)	const Transition* lastTransitionTo()						  const noexcept	{ return lastTransitionTo(stateId<TState>());	}

	/// @brief Get the last transition that caused the current state to be activated
	/// @return Pointer to the last transition that activated the current state
	/// @see `HFSM2_ENABLE_TRANSITION_HISTORY`
	HFSM2_CONSTEXPR(14)	const Transition* lastTransition()							  const noexcept;

#endif

protected:
Core& _core;
StateID _originId = INVALID_STATE_ID;
RegionID _regionId = 0;
};

}
}

namespace hfsm2 {
	namespace detail {

		template <typename TArgs>
		HFSM2_CONSTEXPR(14)
		ControlT<TArgs>::Origin::Origin(ControlT& control_,
		const StateID stateId_) noexcept
	: control{control_}
, prevId{control._originId}
{
	HFSM2_ASSERT(stateId_ < StateList::SIZE);
control._originId = stateId_;
}

template <typename TArgs>
HFSM2_CONSTEXPR(20)
ControlT<TArgs>::Origin::~Origin() noexcept {
control._originId = prevId;
}

template <typename TArgs>
HFSM2_CONSTEXPR(14)
ControlT<TArgs>::Region::Region(ControlT& control_,
								const RegionID regionId_) noexcept
	: control{control_}
	, prevId{control._regionId}
{
	control.setRegion(regionId_);
}

template <typename TArgs>
HFSM2_CONSTEXPR(20)
ControlT<TArgs>::Region::~Region() noexcept {
	control.resetRegion(prevId);
}

template <typename TArgs>
HFSM2_CONSTEXPR(14)
void
ControlT<TArgs>::setRegion(const RegionID regionId_) noexcept {
	HFSM2_ASSERT(_regionId <= regionId_ && regionId_ < RegionList::SIZE);

_regionId = regionId_;
}

template <typename TArgs>
HFSM2_CONSTEXPR(14)
void
ControlT<TArgs>::resetRegion(const RegionID regionId_) noexcept {
	HFSM2_ASSERT(regionId_ <= _regionId && _regionId < RegionList::SIZE);

_regionId = regionId_;
}

#if HFSM2_TRANSITION_HISTORY_AVAILABLE()

template <typename TArgs>
HFSM2_CONSTEXPR(14)
void
ControlT<TArgs>::pinLastTransition(const StateID stateId_,
								   const Short index) noexcept
{
	if (index != INVALID_SHORT) {
		HFSM2_ASSERT(index < TransitionSets::CAPACITY);

		if (!_core.registry.isActive(stateId_))
_core.transitionTargets[stateId_] = index;
	}
}

template <typename TArgs>
HFSM2_CONSTEXPR(14)
const typename ControlT<TArgs>::Transition*
ControlT<TArgs>::lastTransitionTo(const StateID stateId_) const noexcept {
	if (HFSM2_CHECKED(stateId_ < StateList::SIZE)) {
		const Short index = _core.transitionTargets[stateId_];

		if (index < _core.previousTransitions.count())
			return &_core.previousTransitions[index];
	}

	return nullptr;
}

template <typename TArgs>
HFSM2_CONSTEXPR(14)
const typename ControlT<TArgs>::Transition*
ControlT<TArgs>::lastTransition() const noexcept {
	HFSM2_ASSERT(_originId < _core.transitionTargets.CAPACITY);

	return lastTransitionTo(_originId);
}

#endif

}
}

namespace hfsm2 {
	namespace detail {

		template <typename TArgs>
		class PlanControlT
			: public ControlT<TArgs>
		{
			template <typename, typename, typename>
			friend struct S_;

			template <typename, typename, Strategy, typename, typename...>
			friend struct C_;

			template <typename, typename, typename, typename...>
			friend struct O_;

			template <typename, typename>
			friend class R_;

			template <typename, typename>
			friend class RV_;

			protected:
			using Control			= ControlT<TArgs>;

			using typename Control::StateList;
			using typename Control::RegionList;

			using typename Control::Core;

			using TransitionSets	= typename Core::TransitionSets;

#if HFSM2_PLANS_AVAILABLE()
			using typename Control::PlanData;
#endif

			struct Region {
				HFSM2_CONSTEXPR(14)	Region(PlanControlT& control,
				const RegionID regionId_,
				const StateID index,
				const Long size)								noexcept;

				HFSM2_CONSTEXPR(20)	~Region()											noexcept;

				PlanControlT& control;
				const RegionID prevId;
				const Long prevIndex;
				const Long prevSize;
			};

			HFSM2_CONSTEXPR(11)	PlanControlT(Core& core,
			const TransitionSets& currentTransitions)	noexcept
		: Control{core}
	, _currentTransitions{currentTransitions}
{}

	HFSM2_CONSTEXPR(14)	void   setRegion(const RegionID regionId_,
										 const StateID index,
										 const Long size)						noexcept;

	HFSM2_CONSTEXPR(14)	void resetRegion(const RegionID regionId_,
										 const StateID index,
										 const Long size)						noexcept;

public:

#if HFSM2_PLANS_AVAILABLE()
	using typename Control::CPlan;

	using Plan				= PayloadPlanT<TArgs>;

	/// @brief Access plan for the current region
	/// @return Plan for the current region
	/// @see `HFSM2_ENABLE_PLANS`
	HFSM2_CONSTEXPR(14)  Plan plan()										noexcept	{ return  Plan{_core.registry, _core.planData, _regionId							};	}

	/// @brief Access plan for a region
	/// @param `regionId` Region identifier
	/// @return Plan for the region
	/// @see `HFSM2_ENABLE_PLANS`
	HFSM2_CONSTEXPR(14)  Plan plan(const RegionID regionId_)				noexcept	{ return  Plan{_core.registry, _core.planData,  regionId_							};	}

	/// @brief Access plan for a region
	/// @tparam `TRegion` Region head state type
	/// @return Plan for the region
	/// @see `HFSM2_ENABLE_PLANS`
	template <typename TRegion>
	HFSM2_CONSTEXPR(14)  Plan plan()										noexcept	{ return  Plan{_core.registry, _core.planData, Control::template regionId<TRegion>()};	}

	/// @brief Access plan for the current region
	/// @return Plan for the current region
	/// @see `HFSM2_ENABLE_PLANS`
	HFSM2_CONSTEXPR(11)	CPlan plan()								  const noexcept	{ return CPlan{_core.registry, _core.planData, _regionId							};	}

	/// @brief Access plan for a region
	/// @param `regionId`
	/// @return Plan for the region
	/// @see `HFSM2_ENABLE_PLANS`
	HFSM2_CONSTEXPR(11)	CPlan plan(const RegionID regionId_)		  const noexcept	{ return CPlan{_core.registry, _core.planData,  regionId_							};	}

	/// @brief Access plan for a region
	/// @tparam `TRegion` Region head state type
	/// @return Plan for the region
	/// @see `HFSM2_ENABLE_PLANS`
	template <typename TRegion>
	HFSM2_CONSTEXPR(11)	CPlan plan()								  const noexcept	{ return CPlan{_core.registry, _core.planData, Control::template regionId<TRegion>()};	}

#endif

	/// @brief Get current transition requests
	/// @return DynamicArrayT of pending transition requests
	HFSM2_CONSTEXPR(11)	const TransitionSets& currentTransitions()	  const noexcept	{ return _currentTransitions;															}

protected:
	using Control::_core;
using Control::_regionId;

const TransitionSets& _currentTransitions;

StateID _regionStateId = 0;
Long _regionSize = StateList::SIZE;
TaskStatus _taskStatus;
};

}
}

namespace hfsm2 {
	namespace detail {

		template <typename TArgs>
		HFSM2_CONSTEXPR(14)
		PlanControlT<TArgs>::Region::Region(PlanControlT& control_,
		const RegionID regionId_,
		const StateID index,
		const Long size) noexcept
	: control  {control_}
, prevId   {control._regionId}
	, prevIndex{control._regionStateId}
	, prevSize {control._regionSize}
{
	control.setRegion(regionId_, index, size);
}

template <typename TArgs>
HFSM2_CONSTEXPR(20)
PlanControlT<TArgs>::Region::~Region() noexcept {
	control.resetRegion(prevId, prevIndex, prevSize);
}

template <typename TArgs>
HFSM2_CONSTEXPR(14)
void
PlanControlT<TArgs>::setRegion(const RegionID regionId_,
							   const StateID index,
							   const Long size) noexcept
{
	HFSM2_ASSERT(_regionId <= regionId_ && regionId_ <  RegionList::SIZE);
	HFSM2_ASSERT(_regionStateId <= index && index + size <= _regionStateId + _regionSize);

_regionId	   = regionId_;
_regionStateId = index;
_regionSize	   = size;
}

template <typename TArgs>
HFSM2_CONSTEXPR(14)
void
PlanControlT<TArgs>::resetRegion(const RegionID regionId_,
								 const StateID index,
								 const Long size) noexcept
{
	HFSM2_ASSERT(regionId_ <= _regionId && _regionId < RegionList::SIZE);
	HFSM2_ASSERT(index <= _regionStateId && _regionStateId + _regionSize <= index + size);

_regionId	   = regionId_;
_regionStateId = index;
_regionSize	   = size;

	_taskStatus.clear();
}

}
}

namespace hfsm2 {
	namespace detail {

		template <typename TArgs>
		class FullControlBaseT
			: public PlanControlT<TArgs>
		{
			template <typename, typename, typename>
			friend struct S_;

			template <typename, typename, Strategy, typename, typename...>
			friend struct C_;

			template <typename, typename, typename, typename...>
			friend struct O_;

			template <typename, typename>
			friend class R_;

			protected:
			static constexpr Long STATE_COUNT	= TArgs::STATE_COUNT;

			using PlanControl	= PlanControlT<TArgs>;

			using typename PlanControl::StateList;
			using typename PlanControl::RegionList;

			using typename PlanControl::Transition;

#if HFSM2_PLANS_AVAILABLE()
			using TasksBits		= BitArrayT<StateList::SIZE>;
#endif

			struct Lock final {
			HFSM2_CONSTEXPR(14)	 Lock(FullControlBaseT& control_)		noexcept;
			HFSM2_CONSTEXPR(20)	~Lock()									noexcept;

			FullControlBaseT* const control;
		};

		using PlanControl::PlanControl;

		public:
		using PlanControl::context;

		/// @brief Transition into a state
		///   (if transitioning into a region, acts depending on the region type)
		/// @param `stateId` State identifier
		HFSM2_CONSTEXPR(14)	void changeTo (const StateID stateId_)		noexcept;

		/// @brief Transition into a state
		///   (if transitioning into a region, acts depending on the region type)
		/// @tparam `TState` State type
		template <typename TState>
	HFSM2_CONSTEXPR(14)	void changeTo ()							noexcept	{ changeTo (PlanControl::template stateId<TState>());	}

	/// @brief Transition into a state
	///   (if transitioning into a region, activates the initial state)
	/// @param `stateId` State identifier
	HFSM2_CONSTEXPR(14)	void restart  (const StateID stateId_)		noexcept;

	/// @brief Transition into a state
	///   (if transitioning into a region, activates the initial state)
	/// @tparam `TState` State type
	template <typename TState>
HFSM2_CONSTEXPR(14)	void restart  ()							noexcept	{ restart  (PlanControl::template stateId<TState>());	}
```
